LIN {X 55.470,Y -41.308,Z -105.429,A -90.000,B 90.000,C 0.000} C_DIS
LIN {X 55.184,Y -41.308,Z -107.179,A -90.000,B 90.000,C 0.000} C_DIS
LIN {X 54.822,Y -41.308,Z -109.208,A -90.000,B 90.000,C 0.000} C_DIS
LIN {X 54.818,Y -41.308,Z -109.239,A -90.000,B 90.000,C 0.000} C_DIS
LIN {X 54.778,Y -41.308,Z -109.421,A -90.000,B 90.000,C 0.000} C_DIS
LIN {X 54.161,Y -41.308,Z -111.953,A -90.000,B 90.000,C 0.000} C_DIS
LIN {X 54.080,Y -41.308,Z -112.260,A -90.000,B 90.000,C 0.000} C_DIS
LIN {X 53.759,Y -41.308,Z -113.325,A -90.000,B 90.000,C 0.000} C_DIS
LIN {X 53.214,Y -41.308,Z -114.975,A -90.000,B 90.000,C 0.000} C_DIS
LIN {X 52.425,Y -41.308,Z -117.091,A -90.000,B 90.000,C 0.000} C_DIS
LIN {X 52.337,Y -41.308,Z -117.306,A -90.000,B 90.000,C 0.000} C_DIS
LIN {X 51.749,Y -41.308,Z -118.611,A -90.000,B 90.000,C 0.000} C_DIS
LIN {X 50.611,Y -41.308,Z -120.952,A -90.000,B 90.000,C 0.000} C_DIS
LIN {X 50.435,Y -41.308,Z -121.257,A -90.000,B 90.000,C 0.000} C_DIS
LIN {X 50.184,Y -41.308,Z -121.664,A -90.000,B 90.000,C 0.000} C_DIS
LIN {X 48.891,Y -41.308,Z -123.634,A -90.000,B 90.000,C 0.000} C_DIS
LIN {X 48.351,Y -41.308,Z -124.452,A -90.000,B 90.000,C 0.000} C_DIS
LIN {X 48.205,Y -41.308,Z -124.659,A -90.000,B 90.000,C 0.000} C_DIS
LIN {X 47.984,Y -41.308,Z -124.939,A -90.000,B 90.000,C 0.000} C_DIS
LIN {X 45.252,Y -41.308,Z -127.931,A -90.000,B 90.000,C 0.000} C_DIS
LIN {X 44.992,Y -41.308,Z -128.179,A -90.000,B 90.000,C 0.000} C_DIS
LIN {X 44.294,Y -41.308,Z -128.821,A -90.000,B 90.000,C 0.000} C_DIS
LIN {X 41.919,Y -41.308,Z -130.899,A -90.000,B 90.000,C 0.000} C_DIS
LIN {X 40.833,Y -41.308,Z -131.772,A -90.000,B 90.000,C 0.000} C_DIS
LIN {X 38.770,Y -41.308,Z -133.337,A -90.000,B 90.000,C 0.000} C_DIS
LIN {X 37.043,Y -41.308,Z -134.633,A -90.000,B 90.000,C 0.000} C_DIS
LIN {X 35.762,Y -41.308,Z -135.589,A -90.000,B 90.000,C 0.000} C_DIS
LIN {X 35.411,Y -41.308,Z -135.838,A -90.000,B 90.000,C 0.000} C_DIS
LIN {X 33.546,Y -41.308,Z -137.240,A -90.000,B 90.000,C 0.000} C_DIS
LIN {X 32.468,Y -41.308,Z -138.041,A -90.000,B 90.000,C 0.000} C_DIS
LIN {X 32.425,Y -41.308,Z -138.076,A -90.000,B 90.000,C 0.000} C_DIS
LIN {X 29.828,Y -41.308,Z -139.893,A -90.000,B 90.000,C 0.000} C_DIS
LIN {X 29.382,Y -41.308,Z -140.233,A -90.000,B 90.000,C 0.000} C_DIS
LIN {X 26.864,Y -41.308,Z -141.816,A -90.000,B 90.000,C 0.000} C_DIS
LIN {X 26.120,Y -41.308,Z -142.310,A -90.000,B 90.000,C 0.000} C_DIS
LIN {X 25.779,Y -41.308,Z -142.524,A -90.000,B 90.000,C 0.000} C_DIS
LIN {X 22.899,Y -41.308,Z -144.036,A -90.000,B 90.000,C 0.000} C_DIS
LIN {X 21.842,Y -41.308,Z -144.586,A -90.000,B 90.000,C 0.000} C_DIS
LIN {X 21.477,Y -41.308,Z -144.756,A -90.000,B 90.000,C 0.000} C_DIS
LIN {X 18.835,Y -41.308,Z -145.707,A -90.000,B 90.000,C 0.000} C_DIS
LIN {X 16.834,Y -41.308,Z -146.406,A -90.000,B 90.000,C 0.000} C_DIS
LIN {X 15.872,Y -41.308,Z -146.709,A -90.000,B 90.000,C 0.000} C_DIS
LIN {X 11.057,Y -41.308,Z -147.911,A -90.000,B 90.000,C 0.000} C_DIS
LIN {X 10.662,Y -41.308,Z -147.987,A -90.000,B 90.000,C 0.000} C_DIS
LIN {X 9.668,Y -41.308,Z -148.138,A -90.000,B 90.000,C 0.000} C_DIS
LIN {X 7.179,Y -41.308,Z -148.500,A -90.000,B 90.000,C 0.000} C_DIS
LIN {X 6.274,Y -41.308,Z -148.619,A -90.000,B 90.000,C 0.000} C_DIS
LIN {X 5.872,Y -41.308,Z -148.645,A -90.000,B 90.000,C 0.000} C_DIS
LIN {X 3.525,Y -41.308,Z -148.708,A -90.000,B 90.000,C 0.000} C_DIS
LIN {X 1.800,Y -41.308,Z -148.737,A -90.000,B 90.000,C 0.000} C_DIS
LIN {X 1.354,Y -41.308,Z -148.715,A -90.000,B 90.000,C 0.000} C_DIS
LIN {X 0.760,Y -41.308,Z -148.643,A -90.000,B 90.000,C 0.000} C_DIS
LIN {X -2.452,Y -41.308,Z -148.225,A -90.000,B 90.000,C 0.000} C_DIS
LIN {X -2.823,Y -41.308,Z -148.163,A -90.000,B 90.000,C 0.000} C_DIS
LIN {X -3.340,Y -41.308,Z -148.020,A -90.000,B 90.000,C 0.000} C_DIS
LIN {X -6.560,Y -41.308,Z -147.123,A -90.000,B 90.000,C 0.000} C_DIS
LIN {X -6.893,Y -41.308,Z -147.020,A -90.000,B 90.000,C 0.000} C_DIS
LIN {X -6.944,Y -41.308,Z -147.001,A -90.000,B 90.000,C 0.000} C_DIS
LIN {X -10.523,Y -41.308,Z -145.460,A -90.000,B 90.000,C 0.000} C_DIS
LIN {X -10.889,Y -41.308,Z -145.291,A -90.000,B 90.000,C 0.000} C_DIS
LIN {X -14.025,Y -41.308,Z -143.432,A -90.000,B 90.000,C 0.000} C_DIS
LIN {X -14.270,Y -41.308,Z -143.286,A -90.000,B 90.000,C 0.000} C_DIS
LIN {X -14.609,Y -41.308,Z -143.075,A -90.000,B 90.000,C 0.000} C_DIS
LIN {X -16.177,Y -41.308,Z -141.857,A -90.000,B 90.000,C 0.000} C_DIS
LIN {X -16.469,Y -41.308,Z -141.615,A -90.000,B 90.000,C 0.000} C_DIS
LIN {X -17.822,Y -41.308,Z -140.483,A -90.000,B 90.000,C 0.000} C_DIS
LIN {X -18.130,Y -41.308,Z -140.162,A -90.000,B 90.000,C 0.000} C_DIS
LIN {X -19.708,Y -41.308,Z -138.424,A -90.000,B 90.000,C 0.000} C_DIS
LIN {X -20.576,Y -41.308,Z -137.390,A -90.000,B 90.000,C 0.000} C_DIS
LIN {X -21.291,Y -41.308,Z -136.400,A -90.000,B 90.000,C 0.000} C_DIS
LIN {X -21.957,Y -41.308,Z -135.414,A -90.000,B 90.000,C 0.000} C_DIS
LIN {X -22.580,Y -41.308,Z -134.443,A -90.000,B 90.000,C 0.000} C_DIS
LIN {X -22.732,Y -41.308,Z -134.187,A -90.000,B 90.000,C 0.000} C_DIS
LIN {X -22.837,Y -41.308,Z -133.977,A -90.000,B 90.000,C 0.000} C_DIS
LIN {X -23.185,Y -41.308,Z -133.168,A -90.000,B 90.000,C 0.000} C_DIS
LIN {X -23.761,Y -41.308,Z -131.694,A -90.000,B 90.000,C 0.000} C_DIS
LIN {X -24.464,Y -41.308,Z -129.749,A -90.000,B 90.000,C 0.000} C_DIS
LIN {X -25.043,Y -41.308,Z -128.392,A -90.000,B 90.000,C 0.000} C_DIS
LIN {X -25.131,Y -41.308,Z -128.124,A -90.000,B 90.000,C 0.000} C_DIS
LIN {X -25.348,Y -41.308,Z -127.339,A -90.000,B 90.000,C 0.000} C_DIS
LIN {X -25.372,Y -41.308,Z -127.242,A -90.000,B 90.000,C 0.000} C_DIS
LIN {X -25.461,Y -41.308,Z -126.952,A -90.000,B 90.000,C 0.000} C_DIS
LIN {X -25.852,Y -41.308,Z -125.600,A -90.000,B 90.000,C 0.000} C_DIS
LIN {X -26.676,Y -41.308,Z -123.642,A -90.000,B 90.000,C 0.000} C_DIS
LIN {X -26.686,Y -41.308,Z -123.614,A -90.000,B 90.000,C 0.000} C_DIS
LIN {X -27.017,Y -41.308,Z -122.593,A -90.000,B 90.000,C 0.000} C_DIS
LIN {X -27.366,Y -41.308,Z -121.308,A -90.000,B 90.000,C 0.000} C_DIS
LIN {X -28.113,Y -41.308,Z -119.627,A -90.000,B 90.000,C 0.000} C_DIS
LIN {X -28.235,Y -41.308,Z -119.250,A -90.000,B 90.000,C 0.000} C_DIS
LIN {X -28.388,Y -41.308,Z -118.667,A -90.000,B 90.000,C 0.000} C_DIS
LIN {X -28.690,Y -41.308,Z -117.442,A -90.000,B 90.000,C 0.000} C_DIS
LIN {X -29.303,Y -41.308,Z -115.983,A -90.000,B 90.000,C 0.000} C_DIS
LIN {X -29.504,Y -41.308,Z -115.461,A -90.000,B 90.000,C 0.000} C_DIS
LIN {X -29.584,Y -41.308,Z -115.228,A -90.000,B 90.000,C 0.000} C_DIS
LIN {X -29.707,Y -41.308,Z -114.737,A -90.000,B 90.000,C 0.000} C_DIS
LIN {X -29.745,Y -41.308,Z -114.458,A -90.000,B 90.000,C 0.000} C_DIS
LIN {X -29.886,Y -41.308,Z -113.388,A -90.000,B 90.000,C 0.000} C_DIS
LIN {X -30.064,Y -41.308,Z -112.621,A -90.000,B 90.000,C 0.000} C_DIS
LIN {X -30.103,Y -41.308,Z -112.334,A -90.000,B 90.000,C 0.000} C_DIS
LIN {X -30.199,Y -41.308,Z -111.305,A -90.000,B 90.000,C 0.000} C_DIS
LIN {X -30.447,Y -41.308,Z -109.725,A -90.000,B 90.000,C 0.000} C_DIS
LIN {X -30.483,Y -41.308,Z -109.465,A -90.000,B 90.000,C 0.000} C_DIS
LIN {X -30.496,Y -41.308,Z -109.337,A -90.000,B 90.000,C 0.000} C_DIS
LIN {X -30.516,Y -41.308,Z -109.074,A -90.000,B 90.000,C 0.000} C_DIS
LIN {X -30.504,Y -41.308,Z -108.792,A -90.000,B 90.000,C 0.000} C_DIS
LIN {X -30.411,Y -41.308,Z -107.326,A -90.000,B 90.000,C 0.000} C_DIS
LIN {X -30.397,Y -41.308,Z -106.865,A -90.000,B 90.000,C 0.000} C_DIS
LIN {X -30.386,Y -41.308,Z -106.583,A -90.000,B 90.000,C 0.000} C_DIS
LIN {X -30.285,Y -41.308,Z -105.447,A -90.000,B 90.000,C 0.000} C_DIS
LIN {X -30.192,Y -41.308,Z -104.049,A -90.000,B 90.000,C 0.000} C_DIS
LIN {X -30.163,Y -41.308,Z -103.694,A -90.000,B 90.000,C 0.000} C_DIS
LIN {X -30.120,Y -41.308,Z -102.956,A -90.000,B 90.000,C 0.000} C_DIS
LIN {X -29.985,Y -41.308,Z -101.652,A -90.000,B 90.000,C 0.000} C_DIS
LIN {X -29.637,Y -41.308,Z -99.930,A -90.000,B 90.000,C 0.000} C_DIS
LIN {X -29.511,Y -41.308,Z -99.218,A -90.000,B 90.000,C 0.000} C_DIS
LIN {X -29.260,Y -41.308,Z -98.222,A -90.000,B 90.000,C 0.000} C_DIS
LIN {X -28.951,Y -41.308,Z -96.846,A -90.000,B 90.000,C 0.000} C_DIS
LIN {X -28.873,Y -41.308,Z -96.536,A -90.000,B 90.000,C 0.000} C_DIS
LIN {X -28.764,Y -41.308,Z -96.217,A -90.000,B 90.000,C 0.000} C_DIS
LIN {X -28.435,Y -41.308,Z -95.161,A -90.000,B 90.000,C 0.000} C_DIS
LIN {X -28.154,Y -41.308,Z -94.354,A -90.000,B 90.000,C 0.000} C_DIS
LIN {X -28.113,Y -41.308,Z -94.248,A -90.000,B 90.000,C 0.000} C_DIS
LIN {X -28.028,Y -41.308,Z -94.049,A -90.000,B 90.000,C 0.000} C_DIS
LIN {X -27.020,Y -41.308,Z -91.931,A -90.000,B 90.000,C 0.000} C_DIS
LIN {X -26.081,Y -41.308,Z -90.359,A -90.000,B 90.000,C 0.000} C_DIS
LIN {X -25.839,Y -41.308,Z -89.921,A -90.000,B 90.000,C 0.000} C_DIS
LIN {X -25.669,Y -41.308,Z -89.651,A -90.000,B 90.000,C 0.000} C_DIS
LIN {X -24.410,Y -41.308,Z -87.880,A -90.000,B 90.000,C 0.000} C_DIS
LIN {X -24.228,Y -41.308,Z -87.636,A -90.000,B 90.000,C 0.000} C_DIS
LIN {X -23.011,Y -41.308,Z -86.221,A -90.000,B 90.000,C 0.000} C_DIS
LIN {X -22.429,Y -41.308,Z -85.576,A -90.000,B 90.000,C 0.000} C_DIS
LIN {X -22.261,Y -41.308,Z -85.395,A -90.000,B 90.000,C 0.000} C_DIS
LIN {X -21.069,Y -41.308,Z -84.189,A -90.000,B 90.000,C 0.000} C_DIS
LIN {X -20.042,Y -41.308,Z -83.242,A -90.000,B 90.000,C 0.000} C_DIS
LIN {X -19.639,Y -41.308,Z -82.906,A -90.000,B 90.000,C 0.000} C_DIS
LIN {X -19.414,Y -41.308,Z -82.736,A -90.000,B 90.000,C 0.000} C_DIS
LIN {X -18.873,Y -41.308,Z -82.338,A -90.000,B 90.000,C 0.000} C_DIS
LIN {X -17.806,Y -41.308,Z -81.628,A -90.000,B 90.000,C 0.000} C_DIS
LIN {X -16.939,Y -41.308,Z -81.143,A -90.000,B 90.000,C 0.000} C_DIS
LIN {X -16.688,Y -41.308,Z -81.016,A -90.000,B 90.000,C 0.000} C_DIS
LIN {X -15.805,Y -41.308,Z -80.619,A -90.000,B 90.000,C 0.000} C_DIS
LIN {X -14.901,Y -41.308,Z -80.303,A -90.000,B 90.000,C 0.000} C_DIS
LIN {X -13.548,Y -41.308,Z -79.901,A -90.000,B 90.000,C 0.000} C_DIS
LIN {X -12.288,Y -41.308,Z -79.649,A -90.000,B 90.000,C 0.000} C_DIS
LIN {X -12.008,Y -41.308,Z -79.617,A -90.000,B 90.000,C 0.000} C_DIS
LIN {X -11.056,Y -41.308,Z -79.521,A -90.000,B 90.000,C 0.000} C_DIS
LIN {X -10.367,Y -41.308,Z -79.494,A -90.000,B 90.000,C 0.000} C_DIS
LIN {X -8.489,Y -41.308,Z -79.501,A -90.000,B 90.000,C 0.000} C_DIS
LIN {X -5.734,Y -41.308,Z -79.670,A -90.000,B 90.000,C 0.000} C_DIS
LIN {X -5.452,Y -41.308,Z -79.690,A -90.000,B 90.000,C 0.000} C_DIS
LIN {X -4.926,Y -41.308,Z -79.755,A -90.000,B 90.000,C 0.000} C_DIS
LIN {X -3.458,Y -41.308,Z -79.966,A -90.000,B 90.000,C 0.000} C_DIS
LIN {X -2.097,Y -41.308,Z -80.208,A -90.000,B 90.000,C 0.000} C_DIS
LIN {X -1.466,Y -41.308,Z -80.327,A -90.000,B 90.000,C 0.000} C_DIS
LIN {X 0.990,Y -41.308,Z -80.823,A -90.000,B 90.000,C 0.000} C_DIS
LIN {X 2.920,Y -41.308,Z -81.243,A -90.000,B 90.000,C 0.000} C_DIS
LIN {X 3.999,Y -41.308,Z -81.474,A -90.000,B 90.000,C 0.000} C_DIS
LIN {X 6.583,Y -41.308,Z -82.083,A -90.000,B 90.000,C 0.000} C_DIS
LIN {X 7.278,Y -41.308,Z -82.255,A -90.000,B 90.000,C 0.000} C_DIS
LIN {X 9.781,Y -41.308,Z -82.880,A -90.000,B 90.000,C 0.000} C_DIS
LIN {X 10.695,Y -41.308,Z -83.134,A -90.000,B 90.000,C 0.000} C_DIS
LIN {X 12.282,Y -41.308,Z -83.509,A -90.000,B 90.000,C 0.000} C_DIS
LIN {X 12.596,Y -41.308,Z -83.584,A -90.000,B 90.000,C 0.000} C_DIS
LIN {X 13.574,Y -41.308,Z -83.847,A -90.000,B 90.000,C 0.000} C_DIS
LIN {X 14.545,Y -41.308,Z -84.040,A -90.000,B 90.000,C 0.000} C_DIS
LIN {X 16.321,Y -41.308,Z -84.427,A -90.000,B 90.000,C 0.000} C_DIS
LIN {X 16.721,Y -41.308,Z -84.484,A -90.000,B 90.000,C 0.000} C_DIS
LIN {X 17.318,Y -41.308,Z -84.561,A -90.000,B 90.000,C 0.000} C_DIS
LIN {X 18.860,Y -41.308,Z -84.755,A -90.000,B 90.000,C 0.000} C_DIS
LIN {X 19.195,Y -41.308,Z -84.791,A -90.000,B 90.000,C 0.000} C_DIS
LIN {X 20.625,Y -41.308,Z -84.831,A -90.000,B 90.000,C 0.000} C_DIS
LIN {X 21.068,Y -41.308,Z -84.812,A -90.000,B 90.000,C 0.000} C_DIS
LIN {X 21.675,Y -41.308,Z -84.762,A -90.000,B 90.000,C 0.000} C_DIS
LIN {X 22.544,Y -41.308,Z -84.619,A -90.000,B 90.000,C 0.000} C_DIS
LIN {X 22.792,Y -41.308,Z -84.576,A -90.000,B 90.000,C 0.000} C_DIS
LIN {X 23.921,Y -41.308,Z -84.001,A -90.000,B 90.000,C 0.000} C_DIS
LIN {X 24.234,Y -41.308,Z -83.731,A -90.000,B 90.000,C 0.000} C_DIS
LIN {X 25.145,Y -41.308,Z -82.984,A -90.000,B 90.000,C 0.000} C_DIS
LIN {X 26.310,Y -41.308,Z -81.865,A -90.000,B 90.000,C 0.000} C_DIS
LIN {X 26.500,Y -41.308,Z -81.723,A -90.000,B 90.000,C 0.000} C_DIS
LIN {X 27.217,Y -41.308,Z -81.212,A -90.000,B 90.000,C 0.000} C_DIS
LIN {X 27.880,Y -41.308,Z -80.766,A -90.000,B 90.000,C 0.000} C_DIS
LIN {X 28.606,Y -41.308,Z -80.372,A -90.000,B 90.000,C 0.000} C_DIS
LIN {X 28.858,Y -41.308,Z -80.245,A -90.000,B 90.000,C 0.000} C_DIS
LIN {X 32.394,Y -41.308,Z -78.944,A -90.000,B 90.000,C 0.000} C_DIS
LIN {X 34.865,Y -41.308,Z -78.150,A -90.000,B 90.000,C 0.000} C_DIS
LIN {X 36.376,Y -41.308,Z -77.574,A -90.000,B 90.000,C 0.000} C_DIS
LIN {X 36.658,Y -41.308,Z -77.445,A -90.000,B 90.000,C 0.000} C_DIS
LIN {X 36.711,Y -41.308,Z -77.406,A -90.000,B 90.000,C 0.000} C_DIS
LIN {X 36.279,Y -41.308,Z -77.381,A -90.000,B 90.000,C 0.000} C_DIS
LIN {X 35.892,Y -41.308,Z -77.401,A -90.000,B 90.000,C 0.000} C_DIS
LIN {X 35.542,Y -41.308,Z -77.370,A -90.000,B 90.000,C 0.000} C_DIS
LIN {X 34.944,Y -41.308,Z -77.302,A -90.000,B 90.000,C 0.000} C_DIS
LIN {X 34.710,Y -41.308,Z -77.248,A -90.000,B 90.000,C 0.000} C_DIS
LIN {X 34.690,Y -41.308,Z -77.245,A -90.000,B 90.000,C 0.000} C_DIS
LIN {X 34.551,Y -41.308,Z -77.209,A -90.000,B 90.000,C 0.000} C_DIS
LIN {X 34.342,Y -41.308,Z -77.160,A -90.000,B 90.000,C 0.000} C_DIS
LIN {X 34.182,Y -41.308,Z -77.145,A -90.000,B 90.000,C 0.000} C_DIS
LIN {X 33.840,Y -41.308,Z -77.064,A -90.000,B 90.000,C 0.000} C_DIS
LIN {X 33.513,Y -41.308,Z -76.935,A -90.000,B 90.000,C 0.000} C_DIS
LIN {X 33.246,Y -41.308,Z -76.821,A -90.000,B 90.000,C 0.000} C_DIS
LIN {X 33.194,Y -41.308,Z -76.802,A -90.000,B 90.000,C 0.000} C_DIS
LIN {X 32.906,Y -41.308,Z -76.688,A -90.000,B 90.000,C 0.000} C_DIS
LIN {X 32.600,Y -41.308,Z -76.515,A -90.000,B 90.000,C 0.000} C_DIS
LIN {X 32.189,Y -41.308,Z -76.218,A -90.000,B 90.000,C 0.000} C_DIS
LIN {X 32.137,Y -41.308,Z -76.188,A -90.000,B 90.000,C 0.000} C_DIS
LIN {X 32.111,Y -41.308,Z -76.168,A -90.000,B 90.000,C 0.000} C_DIS
LIN {X 31.860,Y -41.308,Z -75.973,A -90.000,B 90.000,C 0.000} C_DIS
LIN {X 31.615,Y -41.308,Z -75.720,A -90.000,B 90.000,C 0.000} C_DIS
LIN {X 31.393,Y -41.308,Z -75.413,A -90.000,B 90.000,C 0.000} C_DIS
LIN {X 31.123,Y -41.308,Z -75.016,A -90.000,B 90.000,C 0.000} C_DIS
LIN {X 30.978,Y -41.308,Z -74.811,A -90.000,B 90.000,C 0.000} C_DIS
LIN {X 30.801,Y -41.308,Z -74.476,A -90.000,B 90.000,C 0.000} C_DIS
LIN {X 30.670,Y -41.308,Z -74.120,A -90.000,B 90.000,C 0.000} C_DIS
LIN {X 30.513,Y -41.308,Z -73.557,A -90.000,B 90.000,C 0.000} C_DIS
LIN {X 30.454,Y -41.308,Z -73.158,A -90.000,B 90.000,C 0.000} C_DIS
LIN {X 30.401,Y -41.308,Z -72.580,A -90.000,B 90.000,C 0.000} C_DIS
LIN {X 30.402,Y -41.308,Z -72.545,A -90.000,B 90.000,C 0.000} C_DIS
LIN {X 30.356,Y -41.308,Z -71.582,A -90.000,B 90.000,C 0.000} C_DIS
LIN {X 30.352,Y -41.308,Z -71.406,A -90.000,B 90.000,C 0.000} C_DIS
LIN {X 30.362,Y -41.308,Z -70.965,A -90.000,B 90.000,C 0.000} C_DIS
LIN {X 30.411,Y -41.308,Z -70.384,A -90.000,B 90.000,C 0.000} C_DIS
LIN {X 30.466,Y -41.308,Z -69.932,A -90.000,B 90.000,C 0.000} C_DIS
LIN {X 30.522,Y -41.308,Z -69.610,A -90.000,B 90.000,C 0.000} C_DIS
LIN {X 30.577,Y -41.308,Z -69.206,A -90.000,B 90.000,C 0.000} C_DIS
LIN {X 30.488,Y -41.308,Z -68.758,A -90.000,B 90.000,C 0.000} C_DIS
LIN {X 30.479,Y -41.308,Z -68.643,A -90.000,B 90.000,C 0.000} C_DIS
LIN {X 30.465,Y -41.308,Z -68.403,A -90.000,B 90.000,C 0.000} C_DIS
LIN {X 30.441,Y -41.308,Z -68.159,A -90.000,B 90.000,C 0.000} C_DIS
LIN {X 30.373,Y -41.308,Z -67.312,A -90.000,B 90.000,C 0.000} C_DIS
LIN {X 30.356,Y -41.308,Z -67.021,A -90.000,B 90.000,C 0.000} C_DIS
LIN {X 30.378,Y -41.308,Z -66.364,A -90.000,B 90.000,C 0.000} C_DIS
LIN {X 30.428,Y -41.308,Z -65.571,A -90.000,B 90.000,C 0.000} C_DIS
LIN {X 30.458,Y -41.308,Z -65.229,A -90.000,B 90.000,C 0.000} C_DIS
LIN {X 30.652,Y -41.308,Z -64.365,A -90.000,B 90.000,C 0.000} C_DIS
LIN {X 30.731,Y -41.308,Z -64.056,A -90.000,B 90.000,C 0.000} C_DIS
LIN {X 30.846,Y -41.308,Z -63.730,A -90.000,B 90.000,C 0.000} C_DIS
LIN {X 30.869,Y -41.308,Z -63.646,A -90.000,B 90.000,C 0.000} C_DIS
LIN {X 30.956,Y -41.308,Z -63.430,A -90.000,B 90.000,C 0.000} C_DIS
LIN {X 31.055,Y -41.308,Z -63.200,A -90.000,B 90.000,C 0.000} C_DIS
LIN {X 31.221,Y -41.308,Z -62.936,A -90.000,B 90.000,C 0.000} C_DIS
LIN {X 31.433,Y -41.308,Z -62.669,A -90.000,B 90.000,C 0.000} C_DIS
LIN {X 31.625,Y -41.308,Z -62.462,A -90.000,B 90.000,C 0.000} C_DIS
LIN {X 31.850,Y -41.308,Z -62.293,A -90.000,B 90.000,C 0.000} C_DIS
LIN {X 31.898,Y -41.308,Z -62.269,A -90.000,B 90.000,C 0.000} C_DIS
LIN {X 31.934,Y -41.308,Z -62.101,A -90.000,B 90.000,C 0.000} C_DIS
LIN {X 32.239,Y -41.308,Z -60.873,A -90.000,B 90.000,C 0.000} C_DIS
LIN {X 32.373,Y -41.308,Z -60.427,A -90.000,B 90.000,C 0.000} C_DIS
LIN {X 32.524,Y -41.308,Z -59.945,A -90.000,B 90.000,C 0.000} C_DIS
LIN {X 32.690,Y -41.308,Z -59.445,A -90.000,B 90.000,C 0.000} C_DIS
LIN {X 32.902,Y -41.308,Z -58.788,A -90.000,B 90.000,C 0.000} C_DIS
LIN {X 33.082,Y -41.308,Z -58.320,A -90.000,B 90.000,C 0.000} C_DIS
LIN {X 33.134,Y -41.308,Z -58.190,A -90.000,B 90.000,C 0.000} C_DIS
LIN {X 33.292,Y -41.308,Z -57.823,A -90.000,B 90.000,C 0.000} C_DIS
LIN {X 33.489,Y -41.308,Z -57.449,A -90.000,B 90.000,C 0.000} C_DIS
LIN {X 33.657,Y -41.308,Z -57.144,A -90.000,B 90.000,C 0.000} C_DIS
LIN {X 33.822,Y -41.308,Z -56.825,A -90.000,B 90.000,C 0.000} C_DIS
LIN {X 33.949,Y -41.308,Z -56.585,A -90.000,B 90.000,C 0.000} C_DIS
LIN {X 34.158,Y -41.308,Z -56.223,A -90.000,B 90.000,C 0.000} C_DIS
LIN {X 34.385,Y -41.308,Z -55.890,A -90.000,B 90.000,C 0.000} C_DIS
LIN {X 34.487,Y -41.308,Z -55.759,A -90.000,B 90.000,C 0.000} C_DIS
LIN {X 34.847,Y -41.308,Z -55.337,A -90.000,B 90.000,C 0.000} C_DIS
LIN {X 34.935,Y -41.308,Z -55.224,A -90.000,B 90.000,C 0.000} C_DIS
LIN {X 35.201,Y -41.308,Z -54.922,A -90.000,B 90.000,C 0.000} C_DIS
LIN {X 35.609,Y -41.308,Z -54.560,A -90.000,B 90.000,C 0.000} C_DIS
LIN {X 35.931,Y -41.308,Z -54.296,A -90.000,B 90.000,C 0.000} C_DIS
LIN {X 36.272,Y -41.308,Z -54.006,A -90.000,B 90.000,C 0.000} C_DIS
LIN {X 36.584,Y -41.308,Z -53.791,A -90.000,B 90.000,C 0.000} C_DIS
LIN {X 36.921,Y -41.308,Z -53.618,A -90.000,B 90.000,C 0.000} C_DIS
LIN {X 37.709,Y -41.308,Z -53.229,A -90.000,B 90.000,C 0.000} C_DIS
LIN {X 38.066,Y -41.308,Z -53.102,A -90.000,B 90.000,C 0.000} C_DIS
LIN {X 38.437,Y -41.308,Z -53.023,A -90.000,B 90.000,C 0.000} C_DIS
LIN {X 38.700,Y -41.308,Z -52.974,A -90.000,B 90.000,C 0.000} C_DIS
LIN {X 39.354,Y -41.308,Z -52.862,A -90.000,B 90.000,C 0.000} C_DIS
LIN {X 39.731,Y -41.308,Z -52.832,A -90.000,B 90.000,C 0.000} C_DIS
LIN {X 40.110,Y -41.308,Z -52.853,A -90.000,B 90.000,C 0.000} C_DIS
LIN {X 41.155,Y -41.308,Z -52.980,A -90.000,B 90.000,C 0.000} C_DIS
LIN {X 41.602,Y -41.308,Z -53.047,A -90.000,B 90.000,C 0.000} C_DIS
LIN {X 41.990,Y -41.308,Z -53.154,A -90.000,B 90.000,C 0.000} C_DIS
LIN {X 42.647,Y -41.308,Z -53.423,A -90.000,B 90.000,C 0.000} C_DIS
LIN {X 42.780,Y -41.308,Z -53.478,A -90.000,B 90.000,C 0.000} C_DIS
LIN {X 43.521,Y -41.308,Z -53.797,A -90.000,B 90.000,C 0.000} C_DIS
LIN {X 44.003,Y -41.308,Z -54.036,A -90.000,B 90.000,C 0.000} C_DIS
LIN {X 44.849,Y -41.308,Z -54.524,A -90.000,B 90.000,C 0.000} C_DIS
LIN {X 45.045,Y -41.308,Z -54.659,A -90.000,B 90.000,C 0.000} C_DIS
LIN {X 45.065,Y -41.308,Z -54.675,A -90.000,B 90.000,C 0.000} C_DIS
LIN {X 45.358,Y -41.308,Z -54.860,A -90.000,B 90.000,C 0.000} C_DIS
LIN {X 45.811,Y -41.308,Z -55.153,A -90.000,B 90.000,C 0.000} C_DIS
LIN {X 46.165,Y -41.308,Z -55.299,A -90.000,B 90.000,C 0.000} C_DIS
LIN {X 46.737,Y -41.308,Z -55.294,A -90.000,B 90.000,C 0.000} C_DIS
LIN {X 47.010,Y -41.308,Z -55.260,A -90.000,B 90.000,C 0.000} C_DIS
LIN {X 47.961,Y -41.308,Z -55.134,A -90.000,B 90.000,C 0.000} C_DIS
LIN {X 48.312,Y -41.308,Z -55.112,A -90.000,B 90.000,C 0.000} C_DIS
LIN {X 48.661,Y -41.308,Z -55.117,A -90.000,B 90.000,C 0.000} C_DIS
LIN {X 49.862,Y -41.308,Z -55.125,A -90.000,B 90.000,C 0.000} C_DIS
LIN {X 50.212,Y -41.308,Z -55.152,A -90.000,B 90.000,C 0.000} C_DIS
LIN {X 50.555,Y -41.308,Z -55.228,A -90.000,B 90.000,C 0.000} C_DIS
LIN {X 50.995,Y -41.308,Z -55.386,A -90.000,B 90.000,C 0.000} C_DIS
LIN {X 52.266,Y -41.308,Z -55.813,A -90.000,B 90.000,C 0.000} C_DIS
LIN {X 52.594,Y -41.308,Z -55.937,A -90.000,B 90.000,C 0.000} C_DIS
LIN {X 52.902,Y -41.308,Z -56.107,A -90.000,B 90.000,C 0.000} C_DIS
LIN {X 53.274,Y -41.308,Z -56.363,A -90.000,B 90.000,C 0.000} C_DIS
LIN {X 54.616,Y -41.308,Z -57.527,A -90.000,B 90.000,C 0.000} C_DIS
LIN {X 55.075,Y -41.308,Z -57.901,A -90.000,B 90.000,C 0.000} C_DIS
LIN {X 55.361,Y -41.308,Z -58.149,A -90.000,B 90.000,C 0.000} C_DIS
LIN {X 55.613,Y -41.308,Z -58.433,A -90.000,B 90.000,C 0.000} C_DIS
LIN {X 56.273,Y -41.308,Z -59.243,A -90.000,B 90.000,C 0.000} C_DIS
LIN {X 56.836,Y -41.308,Z -60.063,A -90.000,B 90.000,C 0.000} C_DIS
LIN {X 57.249,Y -41.308,Z -60.739,A -90.000,B 90.000,C 0.000} C_DIS
LIN {X 57.417,Y -41.308,Z -61.048,A -90.000,B 90.000,C 0.000} C_DIS
LIN {X 57.694,Y -41.308,Z -61.603,A -90.000,B 90.000,C 0.000} C_DIS
LIN {X 58.519,Y -41.308,Z -63.268,A -90.000,B 90.000,C 0.000} C_DIS
LIN {X 58.625,Y -41.308,Z -63.485,A -90.000,B 90.000,C 0.000} C_DIS
LIN {X 58.747,Y -41.308,Z -63.814,A -90.000,B 90.000,C 0.000} C_DIS
LIN {X 58.855,Y -41.308,Z -64.192,A -90.000,B 90.000,C 0.000} C_DIS
LIN {X 59.303,Y -41.308,Z -65.629,A -90.000,B 90.000,C 0.000} C_DIS
LIN {X 59.469,Y -41.308,Z -66.070,A -90.000,B 90.000,C 0.000} C_DIS
LIN {X 59.522,Y -41.308,Z -66.215,A -90.000,B 90.000,C 0.000} C_DIS
LIN {X 59.609,Y -41.308,Z -66.491,A -90.000,B 90.000,C 0.000} C_DIS
LIN {X 59.684,Y -41.308,Z -66.801,A -90.000,B 90.000,C 0.000} C_DIS
LIN {X 59.736,Y -41.308,Z -67.319,A -90.000,B 90.000,C 0.000} C_DIS
LIN {X 59.960,Y -41.308,Z -68.158,A -90.000,B 90.000,C 0.000} C_DIS
LIN {X 59.981,Y -41.308,Z -68.224,A -90.000,B 90.000,C 0.000} C_DIS
LIN {X 60.005,Y -41.308,Z -68.266,A -90.000,B 90.000,C 0.000} C_DIS
LIN {X 60.306,Y -41.308,Z -68.917,A -90.000,B 90.000,C 0.000} C_DIS
LIN {X 60.380,Y -41.308,Z -69.189,A -90.000,B 90.000,C 0.000} C_DIS
LIN {X 60.405,Y -41.308,Z -69.470,A -90.000,B 90.000,C 0.000} C_DIS
LIN {X 60.440,Y -41.308,Z -69.915,A -90.000,B 90.000,C 0.000} C_DIS
LIN {X 60.841,Y -41.308,Z -70.835,A -90.000,B 90.000,C 0.000} C_DIS
LIN {X 61.105,Y -41.308,Z -71.199,A -90.000,B 90.000,C 0.000} C_DIS
LIN {X 61.224,Y -41.308,Z -71.405,A -90.000,B 90.000,C 0.000} C_DIS
LIN {X 61.297,Y -41.308,Z -71.629,A -90.000,B 90.000,C 0.000} C_DIS
LIN {X 61.343,Y -41.308,Z -71.804,A -90.000,B 90.000,C 0.000} C_DIS
LIN {X 61.380,Y -41.308,Z -71.952,A -90.000,B 90.000,C 0.000} C_DIS
LIN {X 61.405,Y -41.308,Z -72.132,A -90.000,B 90.000,C 0.000} C_DIS
LIN {X 61.391,Y -41.308,Z -72.602,A -90.000,B 90.000,C 0.000} C_DIS
LIN {X 61.868,Y -41.308,Z -73.402,A -90.000,B 90.000,C 0.000} C_DIS
LIN {X 61.932,Y -41.308,Z -73.517,A -90.000,B 90.000,C 0.000} C_DIS
LIN {X 63.002,Y -41.308,Z -74.385,A -90.000,B 90.000,C 0.000} C_DIS
LIN {X 63.117,Y -41.308,Z -74.523,A -90.000,B 90.000,C 0.000} C_DIS
LIN {X 63.613,Y -41.308,Z -75.176,A -90.000,B 90.000,C 0.000} C_DIS
LIN {X 65.360,Y -41.308,Z -75.761,A -90.000,B 90.000,C 0.000} C_DIS
LIN {X 66.354,Y -41.308,Z -76.243,A -90.000,B 90.000,C 0.000} C_DIS
LIN {X 66.836,Y -41.308,Z -76.513,A -90.000,B 90.000,C 0.000} C_DIS
LIN {X 67.028,Y -41.308,Z -76.651,A -90.000,B 90.000,C 0.000} C_DIS
LIN {X 67.842,Y -41.308,Z -77.413,A -90.000,B 90.000,C 0.000} C_DIS
LIN {X 68.116,Y -41.308,Z -77.674,A -90.000,B 90.000,C 0.000} C_DIS
LIN {X 69.042,Y -41.308,Z -77.886,A -90.000,B 90.000,C 0.000} C_DIS
LIN {X 69.260,Y -41.308,Z -77.981,A -90.000,B 90.000,C 0.000} C_DIS
LIN {X 69.975,Y -41.308,Z -78.474,A -90.000,B 90.000,C 0.000} C_DIS
LIN {X 70.587,Y -41.308,Z -79.076,A -90.000,B 90.000,C 0.000} C_DIS
LIN {X 70.966,Y -41.308,Z -79.296,A -90.000,B 90.000,C 0.000} C_DIS
LIN {X 71.203,Y -41.308,Z -79.458,A -90.000,B 90.000,C 0.000} C_DIS
LIN {X 71.433,Y -41.308,Z -79.654,A -90.000,B 90.000,C 0.000} C_DIS
LIN {X 71.631,Y -41.308,Z -79.751,A -90.000,B 90.000,C 0.000} C_DIS
LIN {X 71.864,Y -41.308,Z -79.909,A -90.000,B 90.000,C 0.000} C_DIS
LIN {X 72.573,Y -41.308,Z -80.530,A -90.000,B 90.000,C 0.000} C_DIS
LIN {X 72.588,Y -41.308,Z -80.545,A -90.000,B 90.000,C 0.000} C_DIS
LIN {X 72.622,Y -41.308,Z -80.570,A -90.000,B 90.000,C 0.000} C_DIS
LIN {X 72.886,Y -41.308,Z -80.783,A -90.000,B 90.000,C 0.000} C_DIS
LIN {X 73.118,Y -41.308,Z -80.991,A -90.000,B 90.000,C 0.000} C_DIS
LIN {X 73.252,Y -41.308,Z -81.064,A -90.000,B 90.000,C 0.000} C_DIS
LIN {X 73.340,Y -41.308,Z -81.124,A -90.000,B 90.000,C 0.000} C_DIS
LIN {X 73.932,Y -41.308,Z -81.530,A -90.000,B 90.000,C 0.000} C_DIS
LIN {X 74.076,Y -41.308,Z -81.655,A -90.000,B 90.000,C 0.000} C_DIS
LIN {X 74.183,Y -41.308,Z -81.721,A -90.000,B 90.000,C 0.000} C_DIS
LIN {X 74.570,Y -41.308,Z -82.017,A -90.000,B 90.000,C 0.000} C_DIS
LIN {X 74.701,Y -41.308,Z -82.078,A -90.000,B 90.000,C 0.000} C_DIS
LIN {X 75.295,Y -41.308,Z -82.362,A -90.000,B 90.000,C 0.000} C_DIS
LIN {X 75.636,Y -41.308,Z -82.476,A -90.000,B 90.000,C 0.000} C_DIS
LIN {X 76.345,Y -41.308,Z -82.584,A -90.000,B 90.000,C 0.000} C_DIS
LIN {X 76.385,Y -41.308,Z -82.577,A -90.000,B 90.000,C 0.000} C_DIS
LIN {X 77.209,Y -41.308,Z -82.502,A -90.000,B 90.000,C 0.000} C_DIS
LIN {X 77.471,Y -41.308,Z -82.444,A -90.000,B 90.000,C 0.000} C_DIS
LIN {X 78.012,Y -41.308,Z -82.289,A -90.000,B 90.000,C 0.000} C_DIS
LIN {X 78.258,Y -41.308,Z -82.226,A -90.000,B 90.000,C 0.000} C_DIS
LIN {X 78.430,Y -41.308,Z -82.190,A -90.000,B 90.000,C 0.000} C_DIS
LIN {X 79.273,Y -41.308,Z -81.919,A -90.000,B 90.000,C 0.000} C_DIS
LIN {X 79.827,Y -41.308,Z -81.693,A -90.000,B 90.000,C 0.000} C_DIS
LIN {X 79.937,Y -41.308,Z -81.641,A -90.000,B 90.000,C 0.000} C_DIS
LIN {X 80.363,Y -41.308,Z -81.265,A -90.000,B 90.000,C 0.000} C_DIS
LIN {X 80.545,Y -41.308,Z -80.932,A -90.000,B 90.000,C 0.000} C_DIS
LIN {X 80.667,Y -41.308,Z -80.018,A -90.000,B 90.000,C 0.000} C_DIS
LIN {X 80.636,Y -41.308,Z -79.445,A -90.000,B 90.000,C 0.000} C_DIS
LIN {X 80.627,Y -41.308,Z -79.042,A -90.000,B 90.000,C 0.000} C_DIS
LIN {X 80.636,Y -41.308,Z -78.656,A -90.000,B 90.000,C 0.000} C_DIS
LIN {X 80.610,Y -41.308,Z -78.359,A -90.000,B 90.000,C 0.000} C_DIS
LIN {X 80.571,Y -41.308,Z -77.854,A -90.000,B 90.000,C 0.000} C_DIS
LIN {X 80.431,Y -41.308,Z -76.989,A -90.000,B 90.000,C 0.000} C_DIS
LIN {X 80.387,Y -41.308,Z -76.575,A -90.000,B 90.000,C 0.000} C_DIS
LIN {X 80.334,Y -41.308,Z -76.180,A -90.000,B 90.000,C 0.000} C_DIS
LIN {X 80.270,Y -41.308,Z -75.662,A -90.000,B 90.000,C 0.000} C_DIS
LIN {X 80.193,Y -41.308,Z -75.286,A -90.000,B 90.000,C 0.000} C_DIS
LIN {X 80.055,Y -41.308,Z -74.540,A -90.000,B 90.000,C 0.000} C_DIS
LIN {X 80.040,Y -41.308,Z -74.390,A -90.000,B 90.000,C 0.000} C_DIS
LIN {X 79.912,Y -41.308,Z -73.324,A -90.000,B 90.000,C 0.000} C_DIS
LIN {X 79.847,Y -41.308,Z -72.930,A -90.000,B 90.000,C 0.000} C_DIS
LIN {X 79.751,Y -41.308,Z -72.302,A -90.000,B 90.000,C 0.000} C_DIS
LIN {X 79.707,Y -41.308,Z -71.849,A -90.000,B 90.000,C 0.000} C_DIS
LIN {X 79.696,Y -41.308,Z -71.694,A -90.000,B 90.000,C 0.000} C_DIS
LIN {X 79.678,Y -41.308,Z -71.286,A -90.000,B 90.000,C 0.000} C_DIS
LIN {X 79.671,Y -41.308,Z -70.819,A -90.000,B 90.000,C 0.000} C_DIS
LIN {X 79.671,Y -41.308,Z -70.171,A -90.000,B 90.000,C 0.000} C_DIS
LIN {X 79.685,Y -41.308,Z -69.516,A -90.000,B 90.000,C 0.000} C_DIS
LIN {X 79.709,Y -41.308,Z -69.073,A -90.000,B 90.000,C 0.000} C_DIS
LIN {X 79.750,Y -41.308,Z -68.632,A -90.000,B 90.000,C 0.000} C_DIS
LIN {X 79.821,Y -41.308,Z -68.161,A -90.000,B 90.000,C 0.000} C_DIS
LIN {X 79.981,Y -41.308,Z -67.347,A -90.000,B 90.000,C 0.000} C_DIS
LIN {X 80.177,Y -41.308,Z -66.619,A -90.000,B 90.000,C 0.000} C_DIS
LIN {X 80.342,Y -41.308,Z -66.113,A -90.000,B 90.000,C 0.000} C_DIS
LIN {X 80.540,Y -41.308,Z -65.669,A -90.000,B 90.000,C 0.000} C_DIS
LIN {X 81.017,Y -41.308,Z -64.624,A -90.000,B 90.000,C 0.000} C_DIS
LIN {X 81.207,Y -41.308,Z -64.250,A -90.000,B 90.000,C 0.000} C_DIS
LIN {X 81.438,Y -41.308,Z -63.804,A -90.000,B 90.000,C 0.000} C_DIS
LIN {X 81.708,Y -41.308,Z -63.344,A -90.000,B 90.000,C 0.000} C_DIS
LIN {X 82.705,Y -41.308,Z -61.742,A -90.000,B 90.000,C 0.000} C_DIS
LIN {X 84.243,Y -41.308,Z -59.630,A -90.000,B 90.000,C 0.000} C_DIS
LIN {X 85.732,Y -41.308,Z -57.856,A -90.000,B 90.000,C 0.000} C_DIS
LIN {X 86.059,Y -41.308,Z -57.494,A -90.000,B 90.000,C 0.000} C_DIS
LIN {X 87.795,Y -41.308,Z -55.685,A -90.000,B 90.000,C 0.000} C_DIS
LIN {X 89.901,Y -41.308,Z -53.759,A -90.000,B 90.000,C 0.000} C_DIS
LIN {X 90.156,Y -41.308,Z -53.529,A -90.000,B 90.000,C 0.000} C_DIS
LIN {X 92.336,Y -41.308,Z -51.661,A -90.000,B 90.000,C 0.000} C_DIS
LIN {X 94.367,Y -41.308,Z -49.945,A -90.000,B 90.000,C 0.000} C_DIS
LIN {X 96.070,Y -41.308,Z -48.453,A -90.000,B 90.000,C 0.000} C_DIS
LIN {X 97.648,Y -41.308,Z -46.921,A -90.000,B 90.000,C 0.000} C_DIS
LIN {X 99.081,Y -41.308,Z -45.409,A -90.000,B 90.000,C 0.000} C_DIS
LIN {X 100.198,Y -41.308,Z -44.163,A -90.000,B 90.000,C 0.000} C_DIS
LIN {X 101.129,Y -41.308,Z -43.113,A -90.000,B 90.000,C 0.000} C_DIS
LIN {X 101.593,Y -41.308,Z -42.598,A -90.000,B 90.000,C 0.000} C_DIS
LIN {X 102.507,Y -41.308,Z -41.597,A -90.000,B 90.000,C 0.000} C_DIS
LIN {X 103.068,Y -41.308,Z -41.024,A -90.000,B 90.000,C 0.000} C_DIS
LIN {X 103.316,Y -41.308,Z -40.771,A -90.000,B 90.000,C 0.000} C_DIS
LIN {X 103.675,Y -41.308,Z -40.443,A -90.000,B 90.000,C 0.000} C_DIS
LIN {X 103.973,Y -41.308,Z -40.177,A -90.000,B 90.000,C 0.000} C_DIS
LIN {X 104.471,Y -41.308,Z -39.738,A -90.000,B 90.000,C 0.000} C_DIS
LIN {X 104.833,Y -41.308,Z -39.455,A -90.000,B 90.000,C 0.000} C_DIS
LIN {X 105.188,Y -41.308,Z -39.182,A -90.000,B 90.000,C 0.000} C_DIS
LIN {X 105.612,Y -41.308,Z -38.867,A -90.000,B 90.000,C 0.000} C_DIS
LIN {X 105.910,Y -41.308,Z -38.665,A -90.000,B 90.000,C 0.000} C_DIS
LIN {X 106.316,Y -41.308,Z -38.399,A -90.000,B 90.000,C 0.000} C_DIS
LIN {X 106.878,Y -41.308,Z -38.075,A -90.000,B 90.000,C 0.000} C_DIS
LIN {X 107.285,Y -41.308,Z -37.845,A -90.000,B 90.000,C 0.000} C_DIS
LIN {X 107.391,Y -41.308,Z -37.790,A -90.000,B 90.000,C 0.000} C_DIS
LIN {X 108.215,Y -41.308,Z -37.430,A -90.000,B 90.000,C 0.000} C_DIS
LIN {X 108.398,Y -41.308,Z -37.363,A -90.000,B 90.000,C 0.000} C_DIS
LIN {X 108.825,Y -41.308,Z -37.222,A -90.000,B 90.000,C 0.000} C_DIS
LIN {X 109.037,Y -41.308,Z -37.155,A -90.000,B 90.000,C 0.000} C_DIS
LIN {X 109.465,Y -41.308,Z -37.051,A -90.000,B 90.000,C 0.000} C_DIS
LIN {X 109.533,Y -41.308,Z -37.038,A -90.000,B 90.000,C 0.000} C_DIS
LIN {X 110.241,Y -41.308,Z -36.945,A -90.000,B 90.000,C 0.000} C_DIS
LIN {X 110.401,Y -41.308,Z -36.933,A -90.000,B 90.000,C 0.000} C_DIS
LIN {X 110.691,Y -41.308,Z -36.927,A -90.000,B 90.000,C 0.000} C_DIS
LIN {X 111.285,Y -41.308,Z -36.949,A -90.000,B 90.000,C 0.000} C_DIS
LIN {X 111.402,Y -41.308,Z -36.960,A -90.000,B 90.000,C 0.000} C_DIS
LIN {X 111.725,Y -41.308,Z -37.010,A -90.000,B 90.000,C 0.000} C_DIS
LIN {X 111.887,Y -41.308,Z -37.043,A -90.000,B 90.000,C 0.000} C_DIS
LIN {X 112.040,Y -41.308,Z -37.078,A -90.000,B 90.000,C 0.000} C_DIS
LIN {X 112.502,Y -41.308,Z -37.205,A -90.000,B 90.000,C 0.000} C_DIS
LIN {X 112.921,Y -41.308,Z -37.374,A -90.000,B 90.000,C 0.000} C_DIS
LIN {X 113.493,Y -41.308,Z -37.682,A -90.000,B 90.000,C 0.000} C_DIS
LIN {X 113.591,Y -41.308,Z -37.744,A -90.000,B 90.000,C 0.000} C_DIS
LIN {X 113.854,Y -41.308,Z -37.927,A -90.000,B 90.000,C 0.000} C_DIS
LIN {X 113.944,Y -41.308,Z -38.000,A -90.000,B 90.000,C 0.000} C_DIS
LIN {X 114.184,Y -41.308,Z -38.212,A -90.000,B 90.000,C 0.000} C_DIS
LIN {X 114.364,Y -41.308,Z -38.376,A -90.000,B 90.000,C 0.000} C_DIS
LIN {X 114.491,Y -41.308,Z -38.508,A -90.000,B 90.000,C 0.000} C_DIS
LIN {X 114.659,Y -41.308,Z -38.693,A -90.000,B 90.000,C 0.000} C_DIS
LIN {X 114.770,Y -41.308,Z -38.839,A -90.000,B 90.000,C 0.000} C_DIS
LIN {X 114.916,Y -41.308,Z -39.042,A -90.000,B 90.000,C 0.000} C_DIS
LIN {X 115.069,Y -41.308,Z -39.266,A -90.000,B 90.000,C 0.000} C_DIS
LIN {X 115.190,Y -41.308,Z -39.472,A -90.000,B 90.000,C 0.000} C_DIS
LIN {X 115.283,Y -41.308,Z -39.639,A -90.000,B 90.000,C 0.000} C_DIS
LIN {X 115.405,Y -41.308,Z -39.893,A -90.000,B 90.000,C 0.000} C_DIS
LIN {X 115.542,Y -41.308,Z -40.209,A -90.000,B 90.000,C 0.000} C_DIS
LIN {X 115.576,Y -41.308,Z -40.291,A -90.000,B 90.000,C 0.000} C_DIS
LIN {X 115.662,Y -41.308,Z -40.545,A -90.000,B 90.000,C 0.000} C_DIS
LIN {X 115.734,Y -41.308,Z -40.783,A -90.000,B 90.000,C 0.000} C_DIS
LIN {X 115.785,Y -41.308,Z -40.950,A -90.000,B 90.000,C 0.000} C_DIS
LIN {X 115.876,Y -41.308,Z -41.442,A -90.000,B 90.000,C 0.000} C_DIS
LIN {X 115.905,Y -41.308,Z -41.606,A -90.000,B 90.000,C 0.000} C_DIS
LIN {X 115.930,Y -41.308,Z -42.029,A -90.000,B 90.000,C 0.000} C_DIS
LIN {X 115.929,Y -41.308,Z -42.104,A -90.000,B 90.000,C 0.000} C_DIS
LIN {X 115.933,Y -41.308,Z -42.234,A -90.000,B 90.000,C 0.000} C_DIS
LIN {X 115.931,Y -41.308,Z -42.346,A -90.000,B 90.000,C 0.000} C_DIS
LIN {X 115.893,Y -41.308,Z -42.771,A -90.000,B 90.000,C 0.000} C_DIS
LIN {X 115.809,Y -41.308,Z -43.175,A -90.000,B 90.000,C 0.000} C_DIS
LIN {X 115.760,Y -41.308,Z -43.389,A -90.000,B 90.000,C 0.000} C_DIS
LIN {X 115.626,Y -41.308,Z -43.790,A -90.000,B 90.000,C 0.000} C_DIS
LIN {X 115.509,Y -41.308,Z -44.055,A -90.000,B 90.000,C 0.000} C_DIS
LIN {X 115.339,Y -41.308,Z -44.418,A -90.000,B 90.000,C 0.000} C_DIS
LIN {X 115.198,Y -41.308,Z -44.670,A -90.000,B 90.000,C 0.000} C_DIS
LIN {X 115.177,Y -41.308,Z -44.715,A -90.000,B 90.000,C 0.000} C_DIS
LIN {X 115.106,Y -41.308,Z -44.834,A -90.000,B 90.000,C 0.000} C_DIS
LIN {X 115.085,Y -41.308,Z -44.885,A -90.000,B 90.000,C 0.000} C_DIS
LIN {X 115.021,Y -41.308,Z -45.066,A -90.000,B 90.000,C 0.000} C_DIS
LIN {X 114.983,Y -41.308,Z -45.196,A -90.000,B 90.000,C 0.000} C_DIS
LIN {X 114.885,Y -41.308,Z -45.580,A -90.000,B 90.000,C 0.000} C_DIS
LIN {X 114.708,Y -41.308,Z -46.363,A -90.000,B 90.000,C 0.000} C_DIS
LIN {X 114.646,Y -41.308,Z -46.599,A -90.000,B 90.000,C 0.000} C_DIS
LIN {X 114.556,Y -41.308,Z -46.960,A -90.000,B 90.000,C 0.000} C_DIS
LIN {X 114.337,Y -41.308,Z -47.738,A -90.000,B 90.000,C 0.000} C_DIS
LIN {X 114.251,Y -41.308,Z -48.053,A -90.000,B 90.000,C 0.000} C_DIS
LIN {X 114.180,Y -41.308,Z -48.275,A -90.000,B 90.000,C 0.000} C_DIS
LIN {X 114.037,Y -41.308,Z -48.692,A -90.000,B 90.000,C 0.000} C_DIS
LIN {X 113.793,Y -41.308,Z -49.388,A -90.000,B 90.000,C 0.000} C_DIS
LIN {X 113.714,Y -41.308,Z -49.607,A -90.000,B 90.000,C 0.000} C_DIS
LIN {X 113.171,Y -41.308,Z -50.898,A -90.000,B 90.000,C 0.000} C_DIS
LIN {X 112.455,Y -41.308,Z -52.536,A -90.000,B 90.000,C 0.000} C_DIS
LIN {X 111.820,Y -41.308,Z -53.934,A -90.000,B 90.000,C 0.000} C_DIS
LIN {X 111.320,Y -41.308,Z -55.120,A -90.000,B 90.000,C 0.000} C_DIS
LIN {X 111.131,Y -41.308,Z -55.560,A -90.000,B 90.000,C 0.000} C_DIS
LIN {X 110.629,Y -41.308,Z -56.838,A -90.000,B 90.000,C 0.000} C_DIS
LIN {X 110.446,Y -41.308,Z -57.296,A -90.000,B 90.000,C 0.000} C_DIS
LIN {X 109.865,Y -41.308,Z -58.871,A -90.000,B 90.000,C 0.000} C_DIS
LIN {X 109.228,Y -41.308,Z -60.730,A -90.000,B 90.000,C 0.000} C_DIS
LIN {X 108.482,Y -41.308,Z -62.945,A -90.000,B 90.000,C 0.000} C_DIS
LIN {X 108.331,Y -41.308,Z -63.379,A -90.000,B 90.000,C 0.000} C_DIS
LIN {X 107.582,Y -41.308,Z -65.490,A -90.000,B 90.000,C 0.000} C_DIS
LIN {X 106.740,Y -41.308,Z -67.685,A -90.000,B 90.000,C 0.000} C_DIS
LIN {X 105.898,Y -41.308,Z -69.639,A -90.000,B 90.000,C 0.000} C_DIS
LIN {X 105.754,Y -41.308,Z -69.968,A -90.000,B 90.000,C 0.000} C_DIS
LIN {X 105.531,Y -41.308,Z -70.471,A -90.000,B 90.000,C 0.000} C_DIS
LIN {X 104.923,Y -41.308,Z -71.749,A -90.000,B 90.000,C 0.000} C_DIS
LIN {X 104.399,Y -41.308,Z -72.818,A -90.000,B 90.000,C 0.000} C_DIS
LIN {X 104.066,Y -41.308,Z -73.452,A -90.000,B 90.000,C 0.000} C_DIS
LIN {X 103.205,Y -41.308,Z -75.050,A -90.000,B 90.000,C 0.000} C_DIS
LIN {X 102.944,Y -41.308,Z -75.503,A -90.000,B 90.000,C 0.000} C_DIS
LIN {X 101.943,Y -41.308,Z -77.150,A -90.000,B 90.000,C 0.000} C_DIS
LIN {X 101.694,Y -41.308,Z -77.546,A -90.000,B 90.000,C 0.000} C_DIS
LIN {X 100.526,Y -41.308,Z -79.161,A -90.000,B 90.000,C 0.000} C_DIS
LIN {X 100.239,Y -41.308,Z -79.520,A -90.000,B 90.000,C 0.000} C_DIS
LIN {X 99.403,Y -41.308,Z -80.525,A -90.000,B 90.000,C 0.000} C_DIS
LIN {X 98.995,Y -41.308,Z -81.010,A -90.000,B 90.000,C 0.000} C_DIS
LIN {X 97.780,Y -41.308,Z -82.340,A -90.000,B 90.000,C 0.000} C_DIS
LIN {X 97.435,Y -41.308,Z -82.680,A -90.000,B 90.000,C 0.000} C_DIS
LIN {X 96.688,Y -41.308,Z -83.390,A -90.000,B 90.000,C 0.000} C_DIS
LIN {X 96.249,Y -41.308,Z -83.751,A -90.000,B 90.000,C 0.000} C_DIS
LIN {X 95.539,Y -41.308,Z -84.269,A -90.000,B 90.000,C 0.000} C_DIS
LIN {X 94.922,Y -41.308,Z -84.681,A -90.000,B 90.000,C 0.000} C_DIS
LIN {X 93.723,Y -41.308,Z -85.444,A -90.000,B 90.000,C 0.000} C_DIS
LIN {X 93.323,Y -41.308,Z -85.660,A -90.000,B 90.000,C 0.000} C_DIS
LIN {X 92.840,Y -41.308,Z -85.908,A -90.000,B 90.000,C 0.000} C_DIS
LIN {X 92.298,Y -41.308,Z -86.155,A -90.000,B 90.000,C 0.000} C_DIS
LIN {X 91.434,Y -41.308,Z -86.640,A -90.000,B 90.000,C 0.000} C_DIS
LIN {X 91.271,Y -41.308,Z -86.725,A -90.000,B 90.000,C 0.000} C_DIS
LIN {X 90.998,Y -41.308,Z -86.914,A -90.000,B 90.000,C 0.000} C_DIS
LIN {X 90.783,Y -41.308,Z -87.044,A -90.000,B 90.000,C 0.000} C_DIS
LIN {X 90.526,Y -41.308,Z -87.304,A -90.000,B 90.000,C 0.000} C_DIS
LIN {X 90.389,Y -41.308,Z -87.504,A -90.000,B 90.000,C 0.000} C_DIS
LIN {X 90.306,Y -41.308,Z -87.654,A -90.000,B 90.000,C 0.000} C_DIS
LIN {X 90.099,Y -41.308,Z -88.188,A -90.000,B 90.000,C 0.000} C_DIS
LIN {X 89.890,Y -41.308,Z -89.224,A -90.000,B 90.000,C 0.000} C_DIS
LIN {X 89.772,Y -41.308,Z -90.537,A -90.000,B 90.000,C 0.000} C_DIS
LIN {X 89.761,Y -41.308,Z -90.766,A -90.000,B 90.000,C 0.000} C_DIS
LIN {X 89.678,Y -41.308,Z -92.258,A -90.000,B 90.000,C 0.000} C_DIS
LIN {X 89.556,Y -41.308,Z -93.931,A -90.000,B 90.000,C 0.000} C_DIS
LIN {X 89.522,Y -41.308,Z -94.280,A -90.000,B 90.000,C 0.000} C_DIS
LIN {X 89.300,Y -41.308,Z -95.719,A -90.000,B 90.000,C 0.000} C_DIS
LIN {X 89.217,Y -41.308,Z -96.060,A -90.000,B 90.000,C 0.000} C_DIS
LIN {X 88.825,Y -41.308,Z -97.082,A -90.000,B 90.000,C 0.000} C_DIS
LIN {X 88.695,Y -41.308,Z -97.408,A -90.000,B 90.000,C 0.000} C_DIS
LIN {X 88.519,Y -41.308,Z -97.712,A -90.000,B 90.000,C 0.000} C_DIS
LIN {X 87.993,Y -41.308,Z -98.474,A -90.000,B 90.000,C 0.000} C_DIS
LIN {X 87.776,Y -41.308,Z -98.751,A -90.000,B 90.000,C 0.000} C_DIS
LIN {X 87.622,Y -41.308,Z -98.913,A -90.000,B 90.000,C 0.000} C_DIS
LIN {X 87.124,Y -41.308,Z -99.446,A -90.000,B 90.000,C 0.000} C_DIS
LIN {X 86.867,Y -41.308,Z -99.691,A -90.000,B 90.000,C 0.000} C_DIS
LIN {X 86.433,Y -41.308,Z -100.047,A -90.000,B 90.000,C 0.000} C_DIS
LIN {X 85.899,Y -41.308,Z -100.605,A -90.000,B 90.000,C 0.000} C_DIS
LIN {X 85.811,Y -41.308,Z -100.699,A -90.000,B 90.000,C 0.000} C_DIS
LIN {X 85.470,Y -41.308,Z -101.163,A -90.000,B 90.000,C 0.000} C_DIS
LIN {X 85.206,Y -41.308,Z -101.528,A -90.000,B 90.000,C 0.000} C_DIS
LIN {X 85.091,Y -41.308,Z -101.750,A -90.000,B 90.000,C 0.000} C_DIS
LIN {X 84.773,Y -41.308,Z -102.347,A -90.000,B 90.000,C 0.000} C_DIS
LIN {X 84.752,Y -41.308,Z -102.429,A -90.000,B 90.000,C 0.000} C_DIS
LIN {X 84.572,Y -41.308,Z -103.024,A -90.000,B 90.000,C 0.000} C_DIS
LIN {X 84.573,Y -41.308,Z -103.637,A -90.000,B 90.000,C 0.000} C_DIS
LIN {X 84.677,Y -41.308,Z -104.414,A -90.000,B 90.000,C 0.000} C_DIS
LIN {X 84.758,Y -41.308,Z -104.751,A -90.000,B 90.000,C 0.000} C_DIS
LIN {X 84.829,Y -41.308,Z -105.567,A -90.000,B 90.000,C 0.000} C_DIS
LIN {X 84.977,Y -41.308,Z -106.244,A -90.000,B 90.000,C 0.000} C_DIS
LIN {X 85.002,Y -41.308,Z -106.525,A -90.000,B 90.000,C 0.000} C_DIS
LIN {X 84.997,Y -41.308,Z -106.654,A -90.000,B 90.000,C 0.000} C_DIS
LIN {X 84.956,Y -41.308,Z -107.107,A -90.000,B 90.000,C 0.000} C_DIS
LIN {X 84.991,Y -41.308,Z -108.122,A -90.000,B 90.000,C 0.000} C_DIS
LIN {X 84.985,Y -41.308,Z -108.251,A -90.000,B 90.000,C 0.000} C_DIS
LIN {X 84.938,Y -41.308,Z -108.529,A -90.000,B 90.000,C 0.000} C_DIS
LIN {X 84.704,Y -41.308,Z -109.209,A -90.000,B 90.000,C 0.000} C_DIS
LIN {X 84.387,Y -41.308,Z -110.494,A -90.000,B 90.000,C 0.000} C_DIS
LIN {X 84.292,Y -41.308,Z -110.759,A -90.000,B 90.000,C 0.000} C_DIS
LIN {X 83.759,Y -41.308,Z -111.966,A -90.000,B 90.000,C 0.000} C_DIS
LIN {X 83.377,Y -41.308,Z -112.997,A -90.000,B 90.000,C 0.000} C_DIS
LIN {X 82.675,Y -41.308,Z -114.644,A -90.000,B 90.000,C 0.000} C_DIS
LIN {X 82.475,Y -41.308,Z -115.169,A -90.000,B 90.000,C 0.000} C_DIS
LIN {X 81.908,Y -41.308,Z -117.104,A -90.000,B 90.000,C 0.000} C_DIS
LIN {X 81.847,Y -41.308,Z -117.319,A -90.000,B 90.000,C 0.000} C_DIS
LIN {X 81.837,Y -41.308,Z -117.488,A -90.000,B 90.000,C 0.000} C_DIS
LIN {X 81.823,Y -41.308,Z -119.354,A -90.000,B 90.000,C 0.000} C_DIS
LIN {X 82.180,Y -41.308,Z -121.212,A -90.000,B 90.000,C 0.000} C_DIS
LIN {X 82.207,Y -41.308,Z -121.372,A -90.000,B 90.000,C 0.000} C_DIS
LIN {X 82.651,Y -41.308,Z -122.944,A -90.000,B 90.000,C 0.000} C_DIS
LIN {X 82.723,Y -41.308,Z -123.210,A -90.000,B 90.000,C 0.000} C_DIS
LIN {X 82.779,Y -41.308,Z -123.598,A -90.000,B 90.000,C 0.000} C_DIS
LIN {X 83.173,Y -41.308,Z -125.135,A -90.000,B 90.000,C 0.000} C_DIS
LIN {X 83.331,Y -41.308,Z -126.417,A -90.000,B 90.000,C 0.000} C_DIS
LIN {X 83.356,Y -41.308,Z -126.698,A -90.000,B 90.000,C 0.000} C_DIS
LIN {X 83.405,Y -41.308,Z -128.592,A -90.000,B 90.000,C 0.000} C_DIS
LIN {X 83.374,Y -41.308,Z -129.313,A -90.000,B 90.000,C 0.000} C_DIS
LIN {X 83.344,Y -41.308,Z -130.665,A -90.000,B 90.000,C 0.000} C_DIS
LIN {X 83.338,Y -41.308,Z -130.793,A -90.000,B 90.000,C 0.000} C_DIS
LIN {X 83.281,Y -41.308,Z -131.583,A -90.000,B 90.000,C 0.000} C_DIS
LIN {X 83.238,Y -41.308,Z -133.072,A -90.000,B 90.000,C 0.000} C_DIS
LIN {X 83.222,Y -41.308,Z -133.321,A -90.000,B 90.000,C 0.000} C_DIS
LIN {X 83.170,Y -41.308,Z -134.097,A -90.000,B 90.000,C 0.000} C_DIS
LIN {X 83.137,Y -41.308,Z -134.907,A -90.000,B 90.000,C 0.000} C_DIS
LIN {X 83.115,Y -41.308,Z -137.034,A -90.000,B 90.000,C 0.000} C_DIS
LIN {X 83.072,Y -41.308,Z -138.244,A -90.000,B 90.000,C 0.000} C_DIS
LIN {X 83.050,Y -41.308,Z -140.397,A -90.000,B 90.000,C 0.000} C_DIS
LIN {X 82.979,Y -41.308,Z -142.045,A -90.000,B 90.000,C 0.000} C_DIS
LIN {X 82.934,Y -41.308,Z -144.011,A -90.000,B 90.000,C 0.000} C_DIS
LIN {X 82.802,Y -41.308,Z -146.158,A -90.000,B 90.000,C 0.000} C_DIS
LIN {X 82.727,Y -41.308,Z -147.785,A -90.000,B 90.000,C 0.000} C_DIS
LIN {X 82.488,Y -41.308,Z -150.423,A -90.000,B 90.000,C 0.000} C_DIS
LIN {X 82.394,Y -41.308,Z -151.605,A -90.000,B 90.000,C 0.000} C_DIS
LIN {X 82.361,Y -41.308,Z -151.923,A -90.000,B 90.000,C 0.000} C_DIS
LIN {X 81.975,Y -41.308,Z -154.987,A -90.000,B 90.000,C 0.000} C_DIS
LIN {X 81.887,Y -41.308,Z -155.731,A -90.000,B 90.000,C 0.000} C_DIS
LIN {X 81.326,Y -41.308,Z -159.059,A -90.000,B 90.000,C 0.000} C_DIS
LIN {X 81.257,Y -41.308,Z -159.478,A -90.000,B 90.000,C 0.000} C_DIS
LIN {X 80.448,Y -41.308,Z -163.143,A -90.000,B 90.000,C 0.000} C_DIS
LIN {X 80.372,Y -41.308,Z -163.430,A -90.000,B 90.000,C 0.000} C_DIS
LIN {X 79.377,Y -41.308,Z -166.927,A -90.000,B 90.000,C 0.000} C_DIS
LIN {X 78.292,Y -41.308,Z -170.276,A -90.000,B 90.000,C 0.000} C_DIS
LIN {X 77.217,Y -41.308,Z -173.471,A -90.000,B 90.000,C 0.000} C_DIS
LIN {X 76.261,Y -41.308,Z -176.488,A -90.000,B 90.000,C 0.000} C_DIS
LIN {X 75.722,Y -41.308,Z -178.546,A -90.000,B 90.000,C 0.000} C_DIS
LIN {X 75.582,Y -41.308,Z -179.099,A -90.000,B 90.000,C 0.000} C_DIS
LIN {X 75.046,Y -41.308,Z -181.535,A -90.000,B 90.000,C 0.000} C_DIS
LIN {X 74.977,Y -41.308,Z -181.866,A -90.000,B 90.000,C 0.000} C_DIS
LIN {X 74.459,Y -41.308,Z -184.522,A -90.000,B 90.000,C 0.000} C_DIS
LIN {X 74.391,Y -41.308,Z -184.883,A -90.000,B 90.000,C 0.000} C_DIS
LIN {X 73.952,Y -41.308,Z -187.066,A -90.000,B 90.000,C 0.000} C_DIS
LIN {X 73.636,Y -41.308,Z -188.548,A -90.000,B 90.000,C 0.000} C_DIS
LIN {X 73.397,Y -41.308,Z -189.565,A -90.000,B 90.000,C 0.000} C_DIS
LIN {X 73.331,Y -41.308,Z -189.831,A -90.000,B 90.000,C 0.000} C_DIS
LIN {X 72.687,Y -41.308,Z -192.299,A -90.000,B 90.000,C 0.000} C_DIS
LIN {X 72.046,Y -41.308,Z -194.469,A -90.000,B 90.000,C 0.000} C_DIS
LIN {X 71.753,Y -41.308,Z -195.437,A -90.000,B 90.000,C 0.000} C_DIS
LIN {X 70.653,Y -41.308,Z -198.705,A -90.000,B 90.000,C 0.000} C_DIS
LIN {X 70.547,Y -41.308,Z -198.992,A -90.000,B 90.000,C 0.000} C_DIS
LIN {X 69.234,Y -41.308,Z -202.588,A -90.000,B 90.000,C 0.000} C_DIS
LIN {X 69.034,Y -41.308,Z -203.100,A -90.000,B 90.000,C 0.000} C_DIS
LIN {X 67.537,Y -41.308,Z -206.968,A -90.000,B 90.000,C 0.000} C_DIS
LIN {X 67.234,Y -41.308,Z -207.710,A -90.000,B 90.000,C 0.000} C_DIS
LIN {X 65.602,Y -41.308,Z -211.729,A -90.000,B 90.000,C 0.000} C_DIS
LIN {X 65.186,Y -41.308,Z -212.706,A -90.000,B 90.000,C 0.000} C_DIS
LIN {X 63.468,Y -41.308,Z -216.755,A -90.000,B 90.000,C 0.000} C_DIS
LIN {X 61.631,Y -41.308,Z -220.908,A -90.000,B 90.000,C 0.000} C_DIS
LIN {X 61.011,Y -41.308,Z -222.298,A -90.000,B 90.000,C 0.000} C_DIS
LIN {X 58.767,Y -41.308,Z -227.036,A -90.000,B 90.000,C 0.000} C_DIS
LIN {X 58.529,Y -41.308,Z -227.542,A -90.000,B 90.000,C 0.000} C_DIS
LIN {X 56.687,Y -41.308,Z -231.093,A -90.000,B 90.000,C 0.000} C_DIS
LIN {X 55.799,Y -41.308,Z -232.848,A -90.000,B 90.000,C 0.000} C_DIS
LIN {X 53.764,Y -41.308,Z -236.369,A -90.000,B 90.000,C 0.000} C_DIS
LIN {X 52.792,Y -41.308,Z -238.142,A -90.000,B 90.000,C 0.000} C_DIS
LIN {X 51.738,Y -41.308,Z -239.895,A -90.000,B 90.000,C 0.000} C_DIS
LIN {X 51.546,Y -41.308,Z -240.211,A -90.000,B 90.000,C 0.000} C_DIS
LIN {X 49.336,Y -41.308,Z -243.561,A -90.000,B 90.000,C 0.000} C_DIS
LIN {X 49.336,Y -60.000,Z -243.561,A -90.000,B 90.000,C 0.000} C_DIS
LIN {X 26.911,Y -60.000,Z -77.635,A -90.000,B 90.000,C 0.000} C_DIS
LIN {X 26.911,Y -41.308,Z -77.635,A -90.000,B 90.000,C 0.000} C_DIS
LIN {X 26.895,Y -41.308,Z -77.635,A -90.000,B 90.000,C 0.000} C_DIS
LIN {X 25.157,Y -41.308,Z -77.463,A -90.000,B 90.000,C 0.000} C_DIS
LIN {X 24.968,Y -41.308,Z -77.429,A -90.000,B 90.000,C 0.000} C_DIS
LIN {X 24.759,Y -41.308,Z -77.343,A -90.000,B 90.000,C 0.000} C_DIS
LIN {X 23.229,Y -41.308,Z -76.469,A -90.000,B 90.000,C 0.000} C_DIS
LIN {X 23.138,Y -41.308,Z -76.407,A -90.000,B 90.000,C 0.000} C_DIS
LIN {X 23.064,Y -41.308,Z -76.347,A -90.000,B 90.000,C 0.000} C_DIS
LIN {X 22.987,Y -41.308,Z -76.267,A -90.000,B 90.000,C 0.000} C_DIS
LIN {X 22.932,Y -41.308,Z -76.189,A -90.000,B 90.000,C 0.000} C_DIS
LIN {X 22.642,Y -41.308,Z -75.749,A -90.000,B 90.000,C 0.000} C_DIS
LIN {X 22.583,Y -41.308,Z -75.579,A -90.000,B 90.000,C 0.000} C_DIS
LIN {X 22.572,Y -41.308,Z -75.400,A -90.000,B 90.000,C 0.000} C_DIS
LIN {X 22.611,Y -41.308,Z -75.225,A -90.000,B 90.000,C 0.000} C_DIS
LIN {X 22.638,Y -41.308,Z -75.147,A -90.000,B 90.000,C 0.000} C_DIS
LIN {X 22.689,Y -41.308,Z -75.074,A -90.000,B 90.000,C 0.000} C_DIS
LIN {X 22.822,Y -41.308,Z -74.940,A -90.000,B 90.000,C 0.000} C_DIS
LIN {X 22.978,Y -41.308,Z -74.851,A -90.000,B 90.000,C 0.000} C_DIS
LIN {X 23.152,Y -41.308,Z -74.809,A -90.000,B 90.000,C 0.000} C_DIS
LIN {X 23.337,Y -41.308,Z -74.801,A -90.000,B 90.000,C 0.000} C_DIS
LIN {X 23.765,Y -41.308,Z -74.723,A -90.000,B 90.000,C 0.000} C_DIS
LIN {X 23.944,Y -41.308,Z -74.731,A -90.000,B 90.000,C 0.000} C_DIS
LIN {X 24.474,Y -41.308,Z -74.880,A -90.000,B 90.000,C 0.000} C_DIS
LIN {X 24.644,Y -41.308,Z -74.936,A -90.000,B 90.000,C 0.000} C_DIS
LIN {X 25.713,Y -41.308,Z -75.312,A -90.000,B 90.000,C 0.000} C_DIS
LIN {X 25.763,Y -41.308,Z -75.334,A -90.000,B 90.000,C 0.000} C_DIS
LIN {X 26.089,Y -41.308,Z -75.549,A -90.000,B 90.000,C 0.000} C_DIS
LIN {X 26.237,Y -41.308,Z -75.650,A -90.000,B 90.000,C 0.000} C_DIS
LIN {X 26.588,Y -41.308,Z -75.968,A -90.000,B 90.000,C 0.000} C_DIS
LIN {X 27.184,Y -41.308,Z -76.338,A -90.000,B 90.000,C 0.000} C_DIS
LIN {X 27.332,Y -41.308,Z -76.439,A -90.000,B 90.000,C 0.000} C_DIS
LIN {X 27.357,Y -41.308,Z -76.462,A -90.000,B 90.000,C 0.000} C_DIS
LIN {X 27.401,Y -41.308,Z -76.494,A -90.000,B 90.000,C 0.000} C_DIS
LIN {X 27.511,Y -41.308,Z -76.625,A -90.000,B 90.000,C 0.000} C_DIS
LIN {X 27.516,Y -41.308,Z -76.632,A -90.000,B 90.000,C 0.000} C_DIS
LIN {X 27.589,Y -41.308,Z -76.795,A -90.000,B 90.000,C 0.000} C_DIS
LIN {X 27.659,Y -41.308,Z -77.082,A -90.000,B 90.000,C 0.000} C_DIS
LIN {X 27.657,Y -41.308,Z -77.101,A -90.000,B 90.000,C 0.000} C_DIS
LIN {X 27.623,Y -41.308,Z -77.183,A -90.000,B 90.000,C 0.000} C_DIS
LIN {X 27.455,Y -41.308,Z -77.398,A -90.000,B 90.000,C 0.000} C_DIS
LIN {X 27.320,Y -41.308,Z -77.515,A -90.000,B 90.000,C 0.000} C_DIS
LIN {X 27.157,Y -41.308,Z -77.591,A -90.000,B 90.000,C 0.000} C_DIS
LIN {X 27.076,Y -41.308,Z -77.608,A -90.000,B 90.000,C 0.000} C_DIS
LIN {X 26.911,Y -41.308,Z -77.635,A -90.000,B 90.000,C 0.000} C_DIS
LIN {X 26.911,Y -60.000,Z -77.635,A -90.000,B 90.000,C 0.000} C_DIS
LIN {X 59.784,Y -60.000,Z -109.242,A -90.000,B 90.000,C 0.000} C_DIS
LIN {X 59.784,Y -39.308,Z -109.242,A -90.000,B 90.000,C 0.000} C_DIS
LIN {X 58.768,Y -39.308,Z -111.415,A -90.000,B 90.000,C 0.000} C_DIS
LIN {X 58.532,Y -39.308,Z -112.196,A -90.000,B 90.000,C 0.000} C_DIS
LIN {X 58.530,Y -39.308,Z -112.201,A -90.000,B 90.000,C 0.000} C_DIS
LIN {X 58.531,Y -39.308,Z -112.502,A -90.000,B 90.000,C 0.000} C_DIS
LIN {X 58.496,Y -39.308,Z -112.765,A -90.000,B 90.000,C 0.000} C_DIS
LIN {X 59.222,Y -39.308,Z -111.842,A -90.000,B 90.000,C 0.000} C_DIS
LIN {X 59.906,Y -39.308,Z -109.794,A -90.000,B 90.000,C 0.000} C_DIS
LIN {X 60.094,Y -39.308,Z -109.174,A -90.000,B 90.000,C 0.000} C_DIS
LIN {X 59.784,Y -39.308,Z -109.242,A -90.000,B 90.000,C 0.000} C_DIS
LIN {X 59.784,Y -60.000,Z -109.242,A -90.000,B 90.000,C 0.000} C_DIS
LIN {X -80.206,Y -60.000,Z -243.561,A -90.000,B 90.000,C 0.000} C_DIS
LIN {X -80.206,Y -40.663,Z -243.561,A -90.000,B 90.000,C 0.000} C_DIS
LIN {X -80.202,Y -40.649,Z -243.535,A -90.000,B 90.000,C 0.000} C_DIS
LIN {X -80.143,Y -40.540,Z -243.312,A -90.000,B 90.000,C 0.000} C_DIS
LIN {X -80.092,Y -40.478,Z -243.178,A -90.000,B 90.000,C 0.000} C_DIS
LIN {X -80.055,Y -40.443,Z -243.095,A -90.000,B 90.000,C 0.000} C_DIS
LIN {X -79.985,Y -40.389,Z -242.963,A -90.000,B 90.000,C 0.000} C_DIS
LIN {X -79.816,Y -40.299,Z -242.711,A -90.000,B 90.000,C 0.000} C_DIS
LIN {X -79.640,Y -40.242,Z -242.511,A -90.000,B 90.000,C 0.000} C_DIS
LIN {X -79.602,Y -40.233,Z -242.473,A -90.000,B 90.000,C 0.000} C_DIS
LIN {X -79.147,Y -40.187,Z -242.130,A -90.000,B 90.000,C 0.000} C_DIS
LIN {X -77.511,Y -40.188,Z -241.177,A -90.000,B 90.000,C 0.000} C_DIS
LIN {X -74.607,Y -40.211,Z -239.526,A -90.000,B 90.000,C 0.000} C_DIS
LIN {X -72.699,Y -40.211,Z -238.453,A -90.000,B 90.000,C 0.000} C_DIS
LIN {X -71.839,Y -40.204,Z -237.974,A -90.000,B 90.000,C 0.000} C_DIS
LIN {X -71.481,Y -40.203,Z -237.778,A -90.000,B 90.000,C 0.000} C_DIS
LIN {X -68.474,Y -40.218,Z -236.172,A -90.000,B 90.000,C 0.000} C_DIS
LIN {X -63.905,Y -40.218,Z -233.750,A -90.000,B 90.000,C 0.000} C_DIS
LIN {X -62.954,Y -40.209,Z -233.252,A -90.000,B 90.000,C 0.000} C_DIS
LIN {X -59.110,Y -40.208,Z -231.296,A -90.000,B 90.000,C 0.000} C_DIS
LIN {X -56.183,Y -40.219,Z -229.825,A -90.000,B 90.000,C 0.000} C_DIS
LIN {X -54.737,Y -40.217,Z -229.103,A -90.000,B 90.000,C 0.000} C_DIS
LIN {X -53.328,Y -40.217,Z -228.405,A -90.000,B 90.000,C 0.000} C_DIS
LIN {X -51.128,Y -40.223,Z -227.328,A -90.000,B 90.000,C 0.000} C_DIS
LIN {X -50.446,Y -40.227,Z -226.999,A -90.000,B 90.000,C 0.000} C_DIS
LIN {X -47.677,Y -40.236,Z -225.664,A -90.000,B 90.000,C 0.000} C_DIS
LIN {X -45.969,Y -40.253,Z -224.860,A -90.000,B 90.000,C 0.000} C_DIS
LIN {X -44.872,Y -40.260,Z -224.337,A -90.000,B 90.000,C 0.000} C_DIS
LIN {X -42.330,Y -40.273,Z -223.127,A -90.000,B 90.000,C 0.000} C_DIS
LIN {X -40.892,Y -40.288,Z -222.458,A -90.000,B 90.000,C 0.000} C_DIS
LIN {X -39.657,Y -40.295,Z -221.887,A -90.000,B 90.000,C 0.000} C_DIS
LIN {X -39.010,Y -40.295,Z -221.591,A -90.000,B 90.000,C 0.000} C_DIS
LIN {X -37.991,Y -40.303,Z -221.119,A -90.000,B 90.000,C 0.000} C_DIS
LIN {X -37.270,Y -40.303,Z -220.776,A -90.000,B 90.000,C 0.000} C_DIS
LIN {X -35.889,Y -40.307,Z -220.127,A -90.000,B 90.000,C 0.000} C_DIS
LIN {X -34.884,Y -40.316,Z -219.665,A -90.000,B 90.000,C 0.000} C_DIS
LIN {X -33.878,Y -40.322,Z -219.206,A -90.000,B 90.000,C 0.000} C_DIS
LIN {X -32.033,Y -40.342,Z -218.379,A -90.000,B 90.000,C 0.000} C_DIS
LIN {X -31.717,Y -40.347,Z -218.241,A -90.000,B 90.000,C 0.000} C_DIS
LIN {X -30.961,Y -40.368,Z -217.906,A -90.000,B 90.000,C 0.000} C_DIS
LIN {X -27.871,Y -40.408,Z -216.435,A -90.000,B 90.000,C 0.000} C_DIS
LIN {X -27.196,Y -40.414,Z -216.114,A -90.000,B 90.000,C 0.000} C_DIS
LIN {X -25.802,Y -40.424,Z -215.451,A -90.000,B 90.000,C 0.000} C_DIS
LIN {X -24.739,Y -40.439,Z -214.941,A -90.000,B 90.000,C 0.000} C_DIS
LIN {X -23.924,Y -40.439,Z -214.524,A -90.000,B 90.000,C 0.000} C_DIS
LIN {X -21.928,Y -40.429,Z -213.476,A -90.000,B 90.000,C 0.000} C_DIS
LIN {X -20.405,Y -40.453,Z -212.728,A -90.000,B 90.000,C 0.000} C_DIS
LIN {X -19.962,Y -40.466,Z -212.507,A -90.000,B 90.000,C 0.000} C_DIS
LIN {X -19.642,Y -40.477,Z -212.352,A -90.000,B 90.000,C 0.000} C_DIS
LIN {X -18.577,Y -40.490,Z -211.777,A -90.000,B 90.000,C 0.000} C_DIS
LIN {X -16.600,Y -40.530,Z -210.701,A -90.000,B 90.000,C 0.000} C_DIS
LIN {X -15.817,Y -40.539,Z -210.257,A -90.000,B 90.000,C 0.000} C_DIS
LIN {X -15.697,Y -40.541,Z -210.189,A -90.000,B 90.000,C 0.000} C_DIS
LIN {X -15.042,Y -40.560,Z -209.811,A -90.000,B 90.000,C 0.000} C_DIS
LIN {X -14.540,Y -40.570,Z -209.506,A -90.000,B 90.000,C 0.000} C_DIS
LIN {X -13.438,Y -40.575,Z -208.840,A -90.000,B 90.000,C 0.000} C_DIS
LIN {X -12.255,Y -40.571,Z -208.096,A -90.000,B 90.000,C 0.000} C_DIS
LIN {X -11.766,Y -40.567,Z -207.789,A -90.000,B 90.000,C 0.000} C_DIS
LIN {X -10.811,Y -40.575,Z -207.183,A -90.000,B 90.000,C 0.000} C_DIS
LIN {X -8.729,Y -40.569,Z -205.788,A -90.000,B 90.000,C 0.000} C_DIS
LIN {X -8.657,Y -40.569,Z -205.741,A -90.000,B 90.000,C 0.000} C_DIS
LIN {X -7.526,Y -40.587,Z -205.048,A -90.000,B 90.000,C 0.000} C_DIS
LIN {X -6.627,Y -40.619,Z -204.488,A -90.000,B 90.000,C 0.000} C_DIS
LIN {X -5.390,Y -40.625,Z -203.603,A -90.000,B 90.000,C 0.000} C_DIS
LIN {X -3.614,Y -40.645,Z -202.379,A -90.000,B 90.000,C 0.000} C_DIS
LIN {X -2.810,Y -40.671,Z -201.818,A -90.000,B 90.000,C 0.000} C_DIS
LIN {X -0.183,Y -40.662,Z -199.664,A -90.000,B 90.000,C 0.000} C_DIS
LIN {X 0.104,Y -40.662,Z -199.439,A -90.000,B 90.000,C 0.000} C_DIS
LIN {X 0.741,Y -40.682,Z -198.935,A -90.000,B 90.000,C 0.000} C_DIS
LIN {X 3.647,Y -40.638,Z -196.190,A -90.000,B 90.000,C 0.000} C_DIS
LIN {X 3.937,Y -40.641,Z -195.913,A -90.000,B 90.000,C 0.000} C_DIS
LIN {X 4.185,Y -40.647,Z -195.687,A -90.000,B 90.000,C 0.000} C_DIS
LIN {X 4.232,Y -40.647,Z -195.640,A -90.000,B 90.000,C 0.000} C_DIS
LIN {X 6.673,Y -40.593,Z -192.986,A -90.000,B 90.000,C 0.000} C_DIS
LIN {X 7.195,Y -40.590,Z -192.413,A -90.000,B 90.000,C 0.000} C_DIS
LIN {X 7.299,Y -40.590,Z -192.301,A -90.000,B 90.000,C 0.000} C_DIS
LIN {X 9.817,Y -40.531,Z -189.387,A -90.000,B 90.000,C 0.000} C_DIS
LIN {X 10.165,Y -40.530,Z -188.980,A -90.000,B 90.000,C 0.000} C_DIS
LIN {X 12.623,Y -40.470,Z -186.098,A -90.000,B 90.000,C 0.000} C_DIS
LIN {X 13.105,Y -40.467,Z -185.527,A -90.000,B 90.000,C 0.000} C_DIS
LIN {X 13.224,Y -40.462,Z -185.384,A -90.000,B 90.000,C 0.000} C_DIS
LIN {X 15.662,Y -40.409,Z -182.637,A -90.000,B 90.000,C 0.000} C_DIS
LIN {X 15.845,Y -40.409,Z -182.428,A -90.000,B 90.000,C 0.000} C_DIS
LIN {X 15.948,Y -40.404,Z -182.308,A -90.000,B 90.000,C 0.000} C_DIS
LIN {X 16.165,Y -40.393,Z -182.066,A -90.000,B 90.000,C 0.000} C_DIS
LIN {X 16.276,Y -40.390,Z -181.948,A -90.000,B 90.000,C 0.000} C_DIS
LIN {X 18.230,Y -40.361,Z -179.957,A -90.000,B 90.000,C 0.000} C_DIS
LIN {X 18.724,Y -40.353,Z -179.456,A -90.000,B 90.000,C 0.000} C_DIS
LIN {X 18.992,Y -40.349,Z -179.189,A -90.000,B 90.000,C 0.000} C_DIS
LIN {X 19.311,Y -40.349,Z -178.881,A -90.000,B 90.000,C 0.000} C_DIS
LIN {X 21.014,Y -40.335,Z -177.255,A -90.000,B 90.000,C 0.000} C_DIS
LIN {X 21.631,Y -40.328,Z -176.657,A -90.000,B 90.000,C 0.000} C_DIS
LIN {X 22.562,Y -40.315,Z -175.763,A -90.000,B 90.000,C 0.000} C_DIS
LIN {X 22.796,Y -40.314,Z -175.543,A -90.000,B 90.000,C 0.000} C_DIS
LIN {X 23.136,Y -40.318,Z -175.218,A -90.000,B 90.000,C 0.000} C_DIS
LIN {X 24.416,Y -40.303,Z -173.927,A -90.000,B 90.000,C 0.000} C_DIS
LIN {X 24.799,Y -40.312,Z -173.529,A -90.000,B 90.000,C 0.000} C_DIS
LIN {X 25.033,Y -40.310,Z -173.265,A -90.000,B 90.000,C 0.000} C_DIS
LIN {X 26.087,Y -40.292,Z -172.059,A -90.000,B 90.000,C 0.000} C_DIS
LIN {X 26.335,Y -40.297,Z -171.767,A -90.000,B 90.000,C 0.000} C_DIS
LIN {X 26.680,Y -40.288,Z -171.320,A -90.000,B 90.000,C 0.000} C_DIS
LIN {X 27.187,Y -40.280,Z -170.675,A -90.000,B 90.000,C 0.000} C_DIS
LIN {X 27.516,Y -40.274,Z -170.257,A -90.000,B 90.000,C 0.000} C_DIS
LIN {X 27.655,Y -40.274,Z -170.078,A -90.000,B 90.000,C 0.000} C_DIS
LIN {X 28.253,Y -40.257,Z -169.223,A -90.000,B 90.000,C 0.000} C_DIS
LIN {X 28.863,Y -40.245,Z -168.373,A -90.000,B 90.000,C 0.000} C_DIS
LIN {X 29.044,Y -40.246,Z -168.117,A -90.000,B 90.000,C 0.000} C_DIS
LIN {X 29.953,Y -40.221,Z -166.725,A -90.000,B 90.000,C 0.000} C_DIS
LIN {X 30.268,Y -40.216,Z -166.253,A -90.000,B 90.000,C 0.000} C_DIS
LIN {X 30.358,Y -40.217,Z -166.115,A -90.000,B 90.000,C 0.000} C_DIS
LIN {X 30.584,Y -40.207,Z -165.742,A -90.000,B 90.000,C 0.000} C_DIS
LIN {X 31.656,Y -40.173,Z -164.004,A -90.000,B 90.000,C 0.000} C_DIS
LIN {X 31.801,Y -40.173,Z -163.764,A -90.000,B 90.000,C 0.000} C_DIS
LIN {X 32.397,Y -40.149,Z -162.726,A -90.000,B 90.000,C 0.000} C_DIS
LIN {X 32.937,Y -40.132,Z -161.798,A -90.000,B 90.000,C 0.000} C_DIS
LIN {X 33.230,Y -40.133,Z -161.280,A -90.000,B 90.000,C 0.000} C_DIS
LIN {X 33.989,Y -40.113,Z -159.860,A -90.000,B 90.000,C 0.000} C_DIS
LIN {X 34.589,Y -40.123,Z -158.703,A -90.000,B 90.000,C 0.000} C_DIS
LIN {X 34.984,Y -40.117,Z -157.899,A -90.000,B 90.000,C 0.000} C_DIS
LIN {X 35.398,Y -40.133,Z -157.020,A -90.000,B 90.000,C 0.000} C_DIS
LIN {X 35.736,Y -40.151,Z -156.294,A -90.000,B 90.000,C 0.000} C_DIS
LIN {X 35.952,Y -40.153,Z -155.803,A -90.000,B 90.000,C 0.000} C_DIS
LIN {X 36.302,Y -40.190,Z -154.947,A -90.000,B 90.000,C 0.000} C_DIS
LIN {X 36.825,Y -40.225,Z -153.769,A -90.000,B 90.000,C 0.000} C_DIS
LIN {X 36.866,Y -40.227,Z -153.671,A -90.000,B 90.000,C 0.000} C_DIS
LIN {X 36.939,Y -40.237,Z -153.475,A -90.000,B 90.000,C 0.000} C_DIS
LIN {X 37.042,Y -40.253,Z -153.195,A -90.000,B 90.000,C 0.000} C_DIS
LIN {X 37.350,Y -40.267,Z -152.413,A -90.000,B 90.000,C 0.000} C_DIS
LIN {X 37.416,Y -40.272,Z -152.257,A -90.000,B 90.000,C 0.000} C_DIS
LIN {X 37.592,Y -40.295,Z -151.838,A -90.000,B 90.000,C 0.000} C_DIS
LIN {X 37.657,Y -40.302,Z -151.683,A -90.000,B 90.000,C 0.000} C_DIS
LIN {X 37.872,Y -40.314,Z -151.195,A -90.000,B 90.000,C 0.000} C_DIS
LIN {X 38.113,Y -40.341,Z -150.524,A -90.000,B 90.000,C 0.000} C_DIS
LIN {X 38.155,Y -40.347,Z -150.417,A -90.000,B 90.000,C 0.000} C_DIS
LIN {X 38.396,Y -40.386,Z -149.843,A -90.000,B 90.000,C 0.000} C_DIS
LIN {X 38.898,Y -40.401,Z -148.732,A -90.000,B 90.000,C 0.000} C_DIS
LIN {X 39.026,Y -40.422,Z -148.424,A -90.000,B 90.000,C 0.000} C_DIS
LIN {X 39.065,Y -40.428,Z -148.336,A -90.000,B 90.000,C 0.000} C_DIS
LIN {X 39.140,Y -40.440,Z -148.147,A -90.000,B 90.000,C 0.000} C_DIS
LIN {X 39.202,Y -40.450,Z -148.007,A -90.000,B 90.000,C 0.000} C_DIS
LIN {X 39.285,Y -40.454,Z -147.834,A -90.000,B 90.000,C 0.000} C_DIS
LIN {X 39.466,Y -40.458,Z -147.465,A -90.000,B 90.000,C 0.000} C_DIS
LIN {X 39.863,Y -40.456,Z -146.611,A -90.000,B 90.000,C 0.000} C_DIS
LIN {X 39.923,Y -40.460,Z -146.480,A -90.000,B 90.000,C 0.000} C_DIS
LIN {X 40.108,Y -40.474,Z -146.085,A -90.000,B 90.000,C 0.000} C_DIS
LIN {X 40.248,Y -40.486,Z -145.826,A -90.000,B 90.000,C 0.000} C_DIS
LIN {X 40.525,Y -40.486,Z -145.336,A -90.000,B 90.000,C 0.000} C_DIS
LIN {X 40.601,Y -40.483,Z -145.187,A -90.000,B 90.000,C 0.000} C_DIS
LIN {X 41.051,Y -40.503,Z -144.281,A -90.000,B 90.000,C 0.000} C_DIS
LIN {X 41.132,Y -40.507,Z -144.117,A -90.000,B 90.000,C 0.000} C_DIS
LIN {X 41.172,Y -40.509,Z -144.042,A -90.000,B 90.000,C 0.000} C_DIS
LIN {X 41.270,Y -40.518,Z -143.876,A -90.000,B 90.000,C 0.000} C_DIS
LIN {X 41.353,Y -40.518,Z -143.743,A -90.000,B 90.000,C 0.000} C_DIS
LIN {X 42.351,Y -40.510,Z -142.212,A -90.000,B 90.000,C 0.000} C_DIS
LIN {X 42.588,Y -40.516,Z -141.824,A -90.000,B 90.000,C 0.000} C_DIS
LIN {X 42.689,Y -40.516,Z -141.663,A -90.000,B 90.000,C 0.000} C_DIS
LIN {X 42.762,Y -40.517,Z -141.555,A -90.000,B 90.000,C 0.000} C_DIS
LIN {X 43.078,Y -40.516,Z -141.121,A -90.000,B 90.000,C 0.000} C_DIS
LIN {X 43.227,Y -40.512,Z -140.907,A -90.000,B 90.000,C 0.000} C_DIS
LIN {X 44.071,Y -40.522,Z -139.660,A -90.000,B 90.000,C 0.000} C_DIS
LIN {X 44.134,Y -40.524,Z -139.572,A -90.000,B 90.000,C 0.000} C_DIS
LIN {X 45.156,Y -40.514,Z -138.321,A -90.000,B 90.000,C 0.000} C_DIS
LIN {X 45.282,Y -40.516,Z -138.163,A -90.000,B 90.000,C 0.000} C_DIS
LIN {X 45.824,Y -40.524,Z -137.473,A -90.000,B 90.000,C 0.000} C_DIS
LIN {X 46.601,Y -40.526,Z -136.588,A -90.000,B 90.000,C 0.000} C_DIS
LIN {X 47.252,Y -40.518,Z -135.815,A -90.000,B 90.000,C 0.000} C_DIS
LIN {X 47.463,Y -40.520,Z -135.560,A -90.000,B 90.000,C 0.000} C_DIS
LIN {X 47.738,Y -40.525,Z -135.239,A -90.000,B 90.000,C 0.000} C_DIS
LIN {X 48.146,Y -40.526,Z -134.788,A -90.000,B 90.000,C 0.000} C_DIS
LIN {X 48.676,Y -40.534,Z -134.200,A -90.000,B 90.000,C 0.000} C_DIS
LIN {X 49.622,Y -40.553,Z -133.157,A -90.000,B 90.000,C 0.000} C_DIS
LIN {X 50.350,Y -40.576,Z -132.390,A -90.000,B 90.000,C 0.000} C_DIS
LIN {X 52.547,Y -40.577,Z -129.822,A -90.000,B 90.000,C 0.000} C_DIS
LIN {X 53.228,Y -40.630,Z -128.995,A -90.000,B 90.000,C 0.000} C_DIS
LIN {X 54.741,Y -40.638,Z -126.582,A -90.000,B 90.000,C 0.000} C_DIS
LIN {X 55.173,Y -40.637,Z -125.875,A -90.000,B 90.000,C 0.000} C_DIS
LIN {X 55.300,Y -40.634,Z -125.656,A -90.000,B 90.000,C 0.000} C_DIS
LIN {X 56.108,Y -40.638,Z -124.236,A -90.000,B 90.000,C 0.000} C_DIS
LIN {X 56.908,Y -40.623,Z -122.726,A -90.000,B 90.000,C 0.000} C_DIS
LIN {X 57.351,Y -40.609,Z -121.896,A -90.000,B 90.000,C 0.000} C_DIS
LIN {X 57.424,Y -40.610,Z -121.777,A -90.000,B 90.000,C 0.000} C_DIS
LIN {X 57.466,Y -40.608,Z -121.696,A -90.000,B 90.000,C 0.000} C_DIS
LIN {X 57.634,Y -40.605,Z -121.394,A -90.000,B 90.000,C 0.000} C_DIS
LIN {X 59.656,Y -40.599,Z -117.798,A -90.000,B 90.000,C 0.000} C_DIS
LIN {X 59.815,Y -40.593,Z -117.494,A -90.000,B 90.000,C 0.000} C_DIS
LIN {X 60.155,Y -40.588,Z -116.832,A -90.000,B 90.000,C 0.000} C_DIS
LIN {X 60.381,Y -40.587,Z -116.407,A -90.000,B 90.000,C 0.000} C_DIS
LIN {X 61.359,Y -40.570,Z -114.585,A -90.000,B 90.000,C 0.000} C_DIS
LIN {X 61.746,Y -40.563,Z -113.859,A -90.000,B 90.000,C 0.000} C_DIS
LIN {X 62.273,Y -40.559,Z -112.848,A -90.000,B 90.000,C 0.000} C_DIS
LIN {X 62.387,Y -40.553,Z -112.603,A -90.000,B 90.000,C 0.000} C_DIS
LIN {X 63.292,Y -40.519,Z -110.653,A -90.000,B 90.000,C 0.000} C_DIS
LIN {X 63.346,Y -40.516,Z -110.530,A -90.000,B 90.000,C 0.000} C_DIS
LIN {X 63.470,Y -40.514,Z -110.268,A -90.000,B 90.000,C 0.000} C_DIS
LIN {X 64.451,Y -40.521,Z -108.199,A -90.000,B 90.000,C 0.000} C_DIS
LIN {X 64.698,Y -40.532,Z -107.678,A -90.000,B 90.000,C 0.000} C_DIS
LIN {X 65.204,Y -40.547,Z -106.493,A -90.000,B 90.000,C 0.000} C_DIS
LIN {X 65.229,Y -40.546,Z -106.425,A -90.000,B 90.000,C 0.000} C_DIS
LIN {X 65.794,Y -40.573,Z -104.835,A -90.000,B 90.000,C 0.000} C_DIS
LIN {X 65.810,Y -40.578,Z -104.784,A -90.000,B 90.000,C 0.000} C_DIS
LIN {X 65.833,Y -40.584,Z -104.714,A -90.000,B 90.000,C 0.000} C_DIS
LIN {X 66.029,Y -40.620,Z -103.884,A -90.000,B 90.000,C 0.000} C_DIS
LIN {X 66.218,Y -40.657,Z -103.187,A -90.000,B 90.000,C 0.000} C_DIS
LIN {X 66.226,Y -40.658,Z -103.140,A -90.000,B 90.000,C 0.000} C_DIS
LIN {X 66.329,Y -40.669,Z -102.405,A -90.000,B 90.000,C 0.000} C_DIS
LIN {X 66.346,Y -40.682,Z -102.252,A -90.000,B 90.000,C 0.000} C_DIS
LIN {X 66.320,Y -40.705,Z -101.565,A -90.000,B 90.000,C 0.000} C_DIS
LIN {X 66.235,Y -40.688,Z -101.294,A -90.000,B 90.000,C 0.000} C_DIS
LIN {X 65.811,Y -40.679,Z -100.017,A -90.000,B 90.000,C 0.000} C_DIS
LIN {X 65.787,Y -40.677,Z -99.963,A -90.000,B 90.000,C 0.000} C_DIS
LIN {X 65.730,Y -40.670,Z -99.855,A -90.000,B 90.000,C 0.000} C_DIS
LIN {X 65.385,Y -40.654,Z -99.196,A -90.000,B 90.000,C 0.000} C_DIS
LIN {X 65.117,Y -40.648,Z -98.689,A -90.000,B 90.000,C 0.000} C_DIS
LIN {X 64.741,Y -40.642,Z -97.980,A -90.000,B 90.000,C 0.000} C_DIS
LIN {X 64.338,Y -40.647,Z -97.158,A -90.000,B 90.000,C 0.000} C_DIS
LIN {X 64.024,Y -40.635,Z -96.505,A -90.000,B 90.000,C 0.000} C_DIS
LIN {X 63.992,Y -40.634,Z -96.435,A -90.000,B 90.000,C 0.000} C_DIS
LIN {X 63.797,Y -40.632,Z -95.986,A -90.000,B 90.000,C 0.000} C_DIS
LIN {X 63.688,Y -40.629,Z -95.733,A -90.000,B 90.000,C 0.000} C_DIS
LIN {X 63.622,Y -40.629,Z -95.561,A -90.000,B 90.000,C 0.000} C_DIS
LIN {X 63.535,Y -40.633,Z -95.297,A -90.000,B 90.000,C 0.000} C_DIS
LIN {X 63.521,Y -40.635,Z -95.256,A -90.000,B 90.000,C 0.000} C_DIS
LIN {X 63.496,Y -40.636,Z -95.165,A -90.000,B 90.000,C 0.000} C_DIS
LIN {X 63.458,Y -40.641,Z -95.020,A -90.000,B 90.000,C 0.000} C_DIS
LIN {X 63.363,Y -40.651,Z -94.652,A -90.000,B 90.000,C 0.000} C_DIS
LIN {X 63.078,Y -40.664,Z -93.522,A -90.000,B 90.000,C 0.000} C_DIS
LIN {X 63.010,Y -40.654,Z -93.246,A -90.000,B 90.000,C 0.000} C_DIS
LIN {X 62.833,Y -40.600,Z -92.500,A -90.000,B 90.000,C 0.000} C_DIS
LIN {X 62.793,Y -40.589,Z -92.277,A -90.000,B 90.000,C 0.000} C_DIS
LIN {X 62.758,Y -40.580,Z -91.992,A -90.000,B 90.000,C 0.000} C_DIS
LIN {X 62.735,Y -40.581,Z -91.811,A -90.000,B 90.000,C 0.000} C_DIS
LIN {X 62.724,Y -40.582,Z -91.701,A -90.000,B 90.000,C 0.000} C_DIS
LIN {X 62.718,Y -40.586,Z -91.563,A -90.000,B 90.000,C 0.000} C_DIS
LIN {X 62.718,Y -40.588,Z -91.499,A -90.000,B 90.000,C 0.000} C_DIS
LIN {X 62.719,Y -40.586,Z -91.403,A -90.000,B 90.000,C 0.000} C_DIS
LIN {X 62.719,Y -40.576,Z -91.104,A -90.000,B 90.000,C 0.000} C_DIS
LIN {X 62.701,Y -40.591,Z -89.690,A -90.000,B 90.000,C 0.000} C_DIS
LIN {X 62.700,Y -40.587,Z -89.377,A -90.000,B 90.000,C 0.000} C_DIS
LIN {X 62.706,Y -40.539,Z -88.023,A -90.000,B 90.000,C 0.000} C_DIS
LIN {X 62.709,Y -40.536,Z -87.931,A -90.000,B 90.000,C 0.000} C_DIS
LIN {X 62.717,Y -40.538,Z -87.663,A -90.000,B 90.000,C 0.000} C_DIS
LIN {X 62.744,Y -40.545,Z -87.025,A -90.000,B 90.000,C 0.000} C_DIS
LIN {X 62.779,Y -40.576,Z -86.057,A -90.000,B 90.000,C 0.000} C_DIS
LIN {X 62.777,Y -40.577,Z -85.957,A -90.000,B 90.000,C 0.000} C_DIS
LIN {X 62.745,Y -40.585,Z -84.515,A -90.000,B 90.000,C 0.000} C_DIS
LIN {X 62.754,Y -40.595,Z -84.179,A -90.000,B 90.000,C 0.000} C_DIS
LIN {X 62.764,Y -40.602,Z -84.027,A -90.000,B 90.000,C 0.000} C_DIS
LIN {X 62.775,Y -40.608,Z -83.919,A -90.000,B 90.000,C 0.000} C_DIS
LIN {X 62.775,Y -40.611,Z -83.782,A -90.000,B 90.000,C 0.000} C_DIS
LIN {X 62.768,Y -40.635,Z -83.088,A -90.000,B 90.000,C 0.000} C_DIS
LIN {X 62.755,Y -40.677,Z -82.558,A -90.000,B 90.000,C 0.000} C_DIS
LIN {X 62.732,Y -40.694,Z -82.279,A -90.000,B 90.000,C 0.000} C_DIS
LIN {X 62.670,Y -40.747,Z -81.493,A -90.000,B 90.000,C 0.000} C_DIS
LIN {X 62.637,Y -40.772,Z -81.058,A -90.000,B 90.000,C 0.000} C_DIS
LIN {X 62.492,Y -40.771,Z -80.521,A -90.000,B 90.000,C 0.000} C_DIS
LIN {X 62.469,Y -40.772,Z -80.425,A -90.000,B 90.000,C 0.000} C_DIS
LIN {X 62.458,Y -40.773,Z -80.368,A -90.000,B 90.000,C 0.000} C_DIS
LIN {X 62.437,Y -40.785,Z -80.257,A -90.000,B 90.000,C 0.000} C_DIS
LIN {X 62.390,Y -40.823,Z -79.946,A -90.000,B 90.000,C 0.000} C_DIS
LIN {X 62.315,Y -40.909,Z -79.272,A -90.000,B 90.000,C 0.000} C_DIS
LIN {X 62.296,Y -40.939,Z -79.047,A -90.000,B 90.000,C 0.000} C_DIS
LIN {X 62.292,Y -40.980,Z -78.760,A -90.000,B 90.000,C 0.000} C_DIS
LIN {X 62.303,Y -40.999,Z -78.642,A -90.000,B 90.000,C 0.000} C_DIS
LIN {X 62.349,Y -41.062,Z -78.266,A -90.000,B 90.000,C 0.000} C_DIS
LIN {X 62.372,Y -41.087,Z -78.123,A -90.000,B 90.000,C 0.000} C_DIS
LIN {X 62.395,Y -41.105,Z -78.012,A -90.000,B 90.000,C 0.000} C_DIS
LIN {X 62.101,Y -41.122,Z -77.497,A -90.000,B 90.000,C 0.000} C_DIS
LIN {X 62.034,Y -41.113,Z -77.493,A -90.000,B 90.000,C 0.000} C_DIS
LIN {X 61.582,Y -41.082,Z -77.466,A -90.000,B 90.000,C 0.000} C_DIS
LIN {X 61.492,Y -41.077,Z -77.456,A -90.000,B 90.000,C 0.000} C_DIS
LIN {X 61.083,Y -41.051,Z -77.404,A -90.000,B 90.000,C 0.000} C_DIS
LIN {X 60.787,Y -41.036,Z -77.339,A -90.000,B 90.000,C 0.000} C_DIS
LIN {X 60.643,Y -41.015,Z -77.377,A -90.000,B 90.000,C 0.000} C_DIS
LIN {X 60.470,Y -40.991,Z -77.416,A -90.000,B 90.000,C 0.000} C_DIS
LIN {X 60.171,Y -40.955,Z -77.457,A -90.000,B 90.000,C 0.000} C_DIS
LIN {X 59.518,Y -40.887,Z -77.522,A -90.000,B 90.000,C 0.000} C_DIS
LIN {X 59.281,Y -40.875,Z -77.548,A -90.000,B 90.000,C 0.000} C_DIS
LIN {X 59.140,Y -40.870,Z -77.558,A -90.000,B 90.000,C 0.000} C_DIS
LIN {X 59.028,Y -40.868,Z -77.560,A -90.000,B 90.000,C 0.000} C_DIS
LIN {X 58.342,Y -40.860,Z -77.567,A -90.000,B 90.000,C 0.000} C_DIS
LIN {X 57.312,Y -40.805,Z -77.781,A -90.000,B 90.000,C 0.000} C_DIS
LIN {X 56.914,Y -40.794,Z -77.865,A -90.000,B 90.000,C 0.000} C_DIS
LIN {X 56.672,Y -40.788,Z -77.912,A -90.000,B 90.000,C 0.000} C_DIS
LIN {X 55.855,Y -40.799,Z -78.074,A -90.000,B 90.000,C 0.000} C_DIS
LIN {X 55.106,Y -40.780,Z -78.339,A -90.000,B 90.000,C 0.000} C_DIS
LIN {X 54.825,Y -40.773,Z -78.436,A -90.000,B 90.000,C 0.000} C_DIS
LIN {X 54.700,Y -40.771,Z -78.477,A -90.000,B 90.000,C 0.000} C_DIS
LIN {X 53.933,Y -40.800,Z -78.740,A -90.000,B 90.000,C 0.000} C_DIS
LIN {X 52.253,Y -40.865,Z -79.313,A -90.000,B 90.000,C 0.000} C_DIS
LIN {X 51.497,Y -40.896,Z -79.554,A -90.000,B 90.000,C 0.000} C_DIS
LIN {X 50.871,Y -40.911,Z -79.809,A -90.000,B 90.000,C 0.000} C_DIS
LIN {X 50.581,Y -40.949,Z -79.933,A -90.000,B 90.000,C 0.000} C_DIS
LIN {X 49.566,Y -41.070,Z -80.360,A -90.000,B 90.000,C 0.000} C_DIS
LIN {X 49.497,Y -41.083,Z -80.467,A -90.000,B 90.000,C 0.000} C_DIS
LIN {X 49.660,Y -41.083,Z -80.678,A -90.000,B 90.000,C 0.000} C_DIS
LIN {X 49.736,Y -41.080,Z -80.776,A -90.000,B 90.000,C 0.000} C_DIS
LIN {X 49.788,Y -41.076,Z -80.850,A -90.000,B 90.000,C 0.000} C_DIS
LIN {X 49.846,Y -41.070,Z -80.942,A -90.000,B 90.000,C 0.000} C_DIS
LIN {X 49.909,Y -41.062,Z -81.059,A -90.000,B 90.000,C 0.000} C_DIS
LIN {X 50.013,Y -41.049,Z -81.289,A -90.000,B 90.000,C 0.000} C_DIS
LIN {X 50.083,Y -41.041,Z -81.461,A -90.000,B 90.000,C 0.000} C_DIS
LIN {X 50.114,Y -41.037,Z -81.558,A -90.000,B 90.000,C 0.000} C_DIS
LIN {X 50.175,Y -41.030,Z -81.841,A -90.000,B 90.000,C 0.000} C_DIS
LIN {X 50.201,Y -41.028,Z -82.022,A -90.000,B 90.000,C 0.000} C_DIS
LIN {X 50.213,Y -41.027,Z -82.123,A -90.000,B 90.000,C 0.000} C_DIS
LIN {X 50.224,Y -41.027,Z -82.299,A -90.000,B 90.000,C 0.000} C_DIS
LIN {X 50.358,Y -41.009,Z -82.463,A -90.000,B 90.000,C 0.000} C_DIS
LIN {X 50.463,Y -40.995,Z -82.609,A -90.000,B 90.000,C 0.000} C_DIS
LIN {X 50.476,Y -40.995,Z -82.628,A -90.000,B 90.000,C 0.000} C_DIS
LIN {X 50.574,Y -40.993,Z -82.796,A -90.000,B 90.000,C 0.000} C_DIS
LIN {X 51.367,Y -40.994,Z -84.317,A -90.000,B 90.000,C 0.000} C_DIS
LIN {X 51.410,Y -40.992,Z -84.373,A -90.000,B 90.000,C 0.000} C_DIS
LIN {X 52.241,Y -40.930,Z -85.531,A -90.000,B 90.000,C 0.000} C_DIS
LIN {X 52.421,Y -40.928,Z -85.779,A -90.000,B 90.000,C 0.000} C_DIS
LIN {X 52.489,Y -40.928,Z -85.879,A -90.000,B 90.000,C 0.000} C_DIS
LIN {X 52.658,Y -40.928,Z -86.167,A -90.000,B 90.000,C 0.000} C_DIS
LIN {X 53.306,Y -40.930,Z -87.291,A -90.000,B 90.000,C 0.000} C_DIS
LIN {X 53.445,Y -40.924,Z -87.460,A -90.000,B 90.000,C 0.000} C_DIS
LIN {X 53.584,Y -40.920,Z -87.652,A -90.000,B 90.000,C 0.000} C_DIS
LIN {X 53.668,Y -40.919,Z -87.784,A -90.000,B 90.000,C 0.000} C_DIS
LIN {X 54.570,Y -40.874,Z -89.209,A -90.000,B 90.000,C 0.000} C_DIS
LIN {X 54.750,Y -40.872,Z -89.490,A -90.000,B 90.000,C 0.000} C_DIS
LIN {X 54.844,Y -40.872,Z -89.649,A -90.000,B 90.000,C 0.000} C_DIS
LIN {X 54.909,Y -40.870,Z -89.761,A -90.000,B 90.000,C 0.000} C_DIS
LIN {X 54.973,Y -40.868,Z -89.882,A -90.000,B 90.000,C 0.000} C_DIS
LIN {X 55.796,Y -40.891,Z -91.670,A -90.000,B 90.000,C 0.000} C_DIS
LIN {X 55.881,Y -40.886,Z -91.859,A -90.000,B 90.000,C 0.000} C_DIS
LIN {X 55.925,Y -40.883,Z -91.946,A -90.000,B 90.000,C 0.000} C_DIS
LIN {X 56.026,Y -40.878,Z -92.200,A -90.000,B 90.000,C 0.000} C_DIS
LIN {X 56.124,Y -40.877,Z -92.503,A -90.000,B 90.000,C 0.000} C_DIS
LIN {X 56.440,Y -40.880,Z -93.570,A -90.000,B 90.000,C 0.000} C_DIS
LIN {X 56.501,Y -40.882,Z -93.777,A -90.000,B 90.000,C 0.000} C_DIS
LIN {X 56.580,Y -40.884,Z -94.042,A -90.000,B 90.000,C 0.000} C_DIS
LIN {X 56.765,Y -40.862,Z -94.689,A -90.000,B 90.000,C 0.000} C_DIS
LIN {X 57.395,Y -40.787,Z -96.896,A -90.000,B 90.000,C 0.000} C_DIS
LIN {X 57.428,Y -40.784,Z -97.061,A -90.000,B 90.000,C 0.000} C_DIS
LIN {X 57.465,Y -40.783,Z -97.319,A -90.000,B 90.000,C 0.000} C_DIS
LIN {X 57.495,Y -40.783,Z -97.620,A -90.000,B 90.000,C 0.000} C_DIS
LIN {X 57.500,Y -40.785,Z -97.716,A -90.000,B 90.000,C 0.000} C_DIS
LIN {X 57.583,Y -40.788,Z -98.631,A -90.000,B 90.000,C 0.000} C_DIS
LIN {X 57.585,Y -40.787,Z -98.670,A -90.000,B 90.000,C 0.000} C_DIS
LIN {X 57.670,Y -40.741,Z -100.908,A -90.000,B 90.000,C 0.000} C_DIS
LIN {X 57.687,Y -40.721,Z -101.434,A -90.000,B 90.000,C 0.000} C_DIS
LIN {X 57.686,Y -40.716,Z -101.554,A -90.000,B 90.000,C 0.000} C_DIS
LIN {X 57.680,Y -40.710,Z -101.694,A -90.000,B 90.000,C 0.000} C_DIS
LIN {X 57.669,Y -40.703,Z -101.841,A -90.000,B 90.000,C 0.000} C_DIS
LIN {X 57.592,Y -40.677,Z -102.538,A -90.000,B 90.000,C 0.000} C_DIS
LIN {X 57.446,Y -40.667,Z -103.992,A -90.000,B 90.000,C 0.000} C_DIS
LIN {X 57.418,Y -40.661,Z -104.251,A -90.000,B 90.000,C 0.000} C_DIS
LIN {X 57.403,Y -40.654,Z -104.381,A -90.000,B 90.000,C 0.000} C_DIS
LIN {X 57.328,Y -40.573,Z -105.504,A -90.000,B 90.000,C 0.000} C_DIS
LIN {X 57.301,Y -40.562,Z -105.728,A -90.000,B 90.000,C 0.000} C_DIS
LIN {X 57.218,Y -40.549,Z -106.204,A -90.000,B 90.000,C 0.000} C_DIS
LIN {X 57.043,Y -40.541,Z -107.256,A -90.000,B 90.000,C 0.000} C_DIS
LIN {X 57.015,Y -40.535,Z -107.411,A -90.000,B 90.000,C 0.000} C_DIS
LIN {X 56.586,Y -40.457,Z -109.629,A -90.000,B 90.000,C 0.000} C_DIS
LIN {X 56.552,Y -40.454,Z -109.778,A -90.000,B 90.000,C 0.000} C_DIS
LIN {X 56.442,Y -40.449,Z -110.221,A -90.000,B 90.000,C 0.000} C_DIS
LIN {X 55.898,Y -40.411,Z -112.375,A -90.000,B 90.000,C 0.000} C_DIS
LIN {X 55.805,Y -40.408,Z -112.719,A -90.000,B 90.000,C 0.000} C_DIS
LIN {X 55.444,Y -40.386,Z -113.882,A -90.000,B 90.000,C 0.000} C_DIS
LIN {X 54.963,Y -40.365,Z -115.303,A -90.000,B 90.000,C 0.000} C_DIS
LIN {X 54.886,Y -40.361,Z -115.527,A -90.000,B 90.000,C 0.000} C_DIS
LIN {X 54.651,Y -40.357,Z -116.155,A -90.000,B 90.000,C 0.000} C_DIS
LIN {X 54.060,Y -40.330,Z -117.700,A -90.000,B 90.000,C 0.000} C_DIS
LIN {X 53.993,Y -40.329,Z -117.865,A -90.000,B 90.000,C 0.000} C_DIS
LIN {X 53.906,Y -40.330,Z -118.070,A -90.000,B 90.000,C 0.000} C_DIS
LIN {X 53.532,Y -40.318,Z -118.883,A -90.000,B 90.000,C 0.000} C_DIS
LIN {X 53.326,Y -40.304,Z -119.321,A -90.000,B 90.000,C 0.000} C_DIS
LIN {X 52.608,Y -40.278,Z -120.765,A -90.000,B 90.000,C 0.000} C_DIS
LIN {X 52.281,Y -40.271,Z -121.428,A -90.000,B 90.000,C 0.000} C_DIS
LIN {X 52.115,Y -40.261,Z -121.752,A -90.000,B 90.000,C 0.000} C_DIS
LIN {X 51.964,Y -40.261,Z -122.016,A -90.000,B 90.000,C 0.000} C_DIS
LIN {X 51.910,Y -40.259,Z -122.108,A -90.000,B 90.000,C 0.000} C_DIS
LIN {X 51.625,Y -40.246,Z -122.555,A -90.000,B 90.000,C 0.000} C_DIS
LIN {X 50.470,Y -40.222,Z -124.288,A -90.000,B 90.000,C 0.000} C_DIS
LIN {X 49.747,Y -40.193,Z -125.350,A -90.000,B 90.000,C 0.000} C_DIS
LIN {X 49.625,Y -40.190,Z -125.523,A -90.000,B 90.000,C 0.000} C_DIS
LIN {X 49.517,Y -40.186,Z -125.668,A -90.000,B 90.000,C 0.000} C_DIS
LIN {X 49.397,Y -40.185,Z -125.820,A -90.000,B 90.000,C 0.000} C_DIS
LIN {X 49.333,Y -40.181,Z -125.897,A -90.000,B 90.000,C 0.000} C_DIS
LIN {X 49.216,Y -40.175,Z -126.032,A -90.000,B 90.000,C 0.000} C_DIS
LIN {X 46.887,Y -40.138,Z -128.545,A -90.000,B 90.000,C 0.000} C_DIS
LIN {X 46.604,Y -40.130,Z -128.846,A -90.000,B 90.000,C 0.000} C_DIS
LIN {X 46.441,Y -40.122,Z -129.017,A -90.000,B 90.000,C 0.000} C_DIS
LIN {X 46.357,Y -40.120,Z -129.100,A -90.000,B 90.000,C 0.000} C_DIS
LIN {X 46.097,Y -40.110,Z -129.337,A -90.000,B 90.000,C 0.000} C_DIS
LIN {X 45.337,Y -40.088,Z -130.013,A -90.000,B 90.000,C 0.000} C_DIS
LIN {X 43.243,Y -40.061,Z -131.818,A -90.000,B 90.000,C 0.000} C_DIS
LIN {X 42.942,Y -40.047,Z -132.067,A -90.000,B 90.000,C 0.000} C_DIS
LIN {X 41.761,Y -40.027,Z -132.995,A -90.000,B 90.000,C 0.000} C_DIS
LIN {X 39.773,Y -40.007,Z -134.481,A -90.000,B 90.000,C 0.000} C_DIS
LIN {X 37.609,Y -39.967,Z -136.061,A -90.000,B 90.000,C 0.000} C_DIS
LIN {X 36.596,Y -39.938,Z -136.784,A -90.000,B 90.000,C 0.000} C_DIS
LIN {X 36.286,Y -39.938,Z -137.003,A -90.000,B 90.000,C 0.000} C_DIS
LIN {X 34.393,Y -39.899,Z -138.379,A -90.000,B 90.000,C 0.000} C_DIS
LIN {X 33.503,Y -39.883,Z -139.020,A -90.000,B 90.000,C 0.000} C_DIS
LIN {X 33.227,Y -39.879,Z -139.222,A -90.000,B 90.000,C 0.000} C_DIS
LIN {X 32.658,Y -39.881,Z -139.623,A -90.000,B 90.000,C 0.000} C_DIS
LIN {X 30.670,Y -39.858,Z -140.985,A -90.000,B 90.000,C 0.000} C_DIS
LIN {X 30.325,Y -39.846,Z -141.231,A -90.000,B 90.000,C 0.000} C_DIS
LIN {X 30.206,Y -39.840,Z -141.313,A -90.000,B 90.000,C 0.000} C_DIS
LIN {X 30.104,Y -39.838,Z -141.380,A -90.000,B 90.000,C 0.000} C_DIS
LIN {X 29.038,Y -39.842,Z -142.056,A -90.000,B 90.000,C 0.000} C_DIS
LIN {X 27.597,Y -39.834,Z -142.951,A -90.000,B 90.000,C 0.000} C_DIS
LIN {X 26.950,Y -39.819,Z -143.362,A -90.000,B 90.000,C 0.000} C_DIS
LIN {X 26.698,Y -39.815,Z -143.518,A -90.000,B 90.000,C 0.000} C_DIS
LIN {X 26.480,Y -39.805,Z -143.642,A -90.000,B 90.000,C 0.000} C_DIS
LIN {X 26.392,Y -39.804,Z -143.690,A -90.000,B 90.000,C 0.000} C_DIS
LIN {X 24.352,Y -39.811,Z -144.770,A -90.000,B 90.000,C 0.000} C_DIS
LIN {X 22.834,Y -39.820,Z -145.576,A -90.000,B 90.000,C 0.000} C_DIS
LIN {X 22.635,Y -39.819,Z -145.678,A -90.000,B 90.000,C 0.000} C_DIS
LIN {X 22.456,Y -39.816,Z -145.767,A -90.000,B 90.000,C 0.000} C_DIS
LIN {X 22.256,Y -39.817,Z -145.863,A -90.000,B 90.000,C 0.000} C_DIS
LIN {X 22.039,Y -39.816,Z -145.962,A -90.000,B 90.000,C 0.000} C_DIS
LIN {X 21.929,Y -39.818,Z -146.010,A -90.000,B 90.000,C 0.000} C_DIS
LIN {X 21.754,Y -39.825,Z -146.082,A -90.000,B 90.000,C 0.000} C_DIS
LIN {X 21.166,Y -39.840,Z -146.311,A -90.000,B 90.000,C 0.000} C_DIS
LIN {X 19.940,Y -39.863,Z -146.779,A -90.000,B 90.000,C 0.000} C_DIS
LIN {X 19.289,Y -39.859,Z -147.008,A -90.000,B 90.000,C 0.000} C_DIS
LIN {X 18.452,Y -39.857,Z -147.298,A -90.000,B 90.000,C 0.000} C_DIS
LIN {X 17.955,Y -39.854,Z -147.469,A -90.000,B 90.000,C 0.000} C_DIS
LIN {X 17.327,Y -39.848,Z -147.682,A -90.000,B 90.000,C 0.000} C_DIS
LIN {X 16.996,Y -39.850,Z -147.790,A -90.000,B 90.000,C 0.000} C_DIS
LIN {X 16.265,Y -39.850,Z -148.020,A -90.000,B 90.000,C 0.000} C_DIS
LIN {X 15.173,Y -39.884,Z -148.330,A -90.000,B 90.000,C 0.000} C_DIS
LIN {X 14.231,Y -39.910,Z -148.592,A -90.000,B 90.000,C 0.000} C_DIS
LIN {X 13.439,Y -39.914,Z -148.794,A -90.000,B 90.000,C 0.000} C_DIS
LIN {X 12.800,Y -39.911,Z -148.951,A -90.000,B 90.000,C 0.000} C_DIS
LIN {X 11.387,Y -39.894,Z -149.286,A -90.000,B 90.000,C 0.000} C_DIS
LIN {X 10.876,Y -39.902,Z -149.392,A -90.000,B 90.000,C 0.000} C_DIS
LIN {X 9.877,Y -39.938,Z -149.579,A -90.000,B 90.000,C 0.000} C_DIS
LIN {X 9.402,Y -39.950,Z -149.659,A -90.000,B 90.000,C 0.000} C_DIS
LIN {X 8.997,Y -39.951,Z -149.719,A -90.000,B 90.000,C 0.000} C_DIS
LIN {X 7.388,Y -39.933,Z -149.936,A -90.000,B 90.000,C 0.000} C_DIS
LIN {X 7.054,Y -39.931,Z -149.979,A -90.000,B 90.000,C 0.000} C_DIS
LIN {X 6.442,Y -39.922,Z -150.051,A -90.000,B 90.000,C 0.000} C_DIS
LIN {X 5.965,Y -39.931,Z -150.092,A -90.000,B 90.000,C 0.000} C_DIS
LIN {X 5.265,Y -39.959,Z -150.138,A -90.000,B 90.000,C 0.000} C_DIS
LIN {X 4.869,Y -39.966,Z -150.155,A -90.000,B 90.000,C 0.000} C_DIS
LIN {X 3.721,Y -39.957,Z -150.177,A -90.000,B 90.000,C 0.000} C_DIS
LIN {X 1.825,Y -39.930,Z -150.185,A -90.000,B 90.000,C 0.000} C_DIS
LIN {X 1.731,Y -39.930,Z -150.184,A -90.000,B 90.000,C 0.000} C_DIS
LIN {X 1.284,Y -39.939,Z -150.171,A -90.000,B 90.000,C 0.000} C_DIS
LIN {X 1.197,Y -39.942,Z -150.167,A -90.000,B 90.000,C 0.000} C_DIS
LIN {X 0.800,Y -39.954,Z -150.131,A -90.000,B 90.000,C 0.000} C_DIS
LIN {X 0.222,Y -39.952,Z -150.056,A -90.000,B 90.000,C 0.000} C_DIS
LIN {X -2.689,Y -39.924,Z -149.649,A -90.000,B 90.000,C 0.000} C_DIS
LIN {X -2.815,Y -39.925,Z -149.629,A -90.000,B 90.000,C 0.000} C_DIS
LIN {X -3.060,Y -39.923,Z -149.586,A -90.000,B 90.000,C 0.000} C_DIS
LIN {X -3.211,Y -39.925,Z -149.555,A -90.000,B 90.000,C 0.000} C_DIS
LIN {X -4.062,Y -39.924,Z -149.317,A -90.000,B 90.000,C 0.000} C_DIS
LIN {X -6.966,Y -39.916,Z -148.499,A -90.000,B 90.000,C 0.000} C_DIS
LIN {X -7.197,Y -39.917,Z -148.430,A -90.000,B 90.000,C 0.000} C_DIS
LIN {X -7.300,Y -39.912,Z -148.393,A -90.000,B 90.000,C 0.000} C_DIS
LIN {X -7.442,Y -39.908,Z -148.338,A -90.000,B 90.000,C 0.000} C_DIS
LIN {X -9.169,Y -39.920,Z -147.610,A -90.000,B 90.000,C 0.000} C_DIS
LIN {X -11.038,Y -39.930,Z -146.816,A -90.000,B 90.000,C 0.000} C_DIS
LIN {X -11.202,Y -39.931,Z -146.744,A -90.000,B 90.000,C 0.000} C_DIS
LIN {X -11.491,Y -39.918,Z -146.597,A -90.000,B 90.000,C 0.000} C_DIS
LIN {X -11.621,Y -39.917,Z -146.527,A -90.000,B 90.000,C 0.000} C_DIS
LIN {X -14.581,Y -39.970,Z -144.831,A -90.000,B 90.000,C 0.000} C_DIS
LIN {X -15.102,Y -39.976,Z -144.525,A -90.000,B 90.000,C 0.000} C_DIS
LIN {X -15.225,Y -39.970,Z -144.442,A -90.000,B 90.000,C 0.000} C_DIS
LIN {X -15.516,Y -39.961,Z -144.242,A -90.000,B 90.000,C 0.000} C_DIS
LIN {X -17.104,Y -39.998,Z -143.050,A -90.000,B 90.000,C 0.000} C_DIS
LIN {X -17.898,Y -40.021,Z -142.415,A -90.000,B 90.000,C 0.000} C_DIS
LIN {X -18.395,Y -40.035,Z -142.013,A -90.000,B 90.000,C 0.000} C_DIS
LIN {X -18.707,Y -40.038,Z -141.756,A -90.000,B 90.000,C 0.000} C_DIS
LIN {X -18.810,Y -40.034,Z -141.665,A -90.000,B 90.000,C 0.000} C_DIS
LIN {X -18.932,Y -40.034,Z -141.551,A -90.000,B 90.000,C 0.000} C_DIS
LIN {X -19.248,Y -40.046,Z -141.238,A -90.000,B 90.000,C 0.000} C_DIS
LIN {X -19.947,Y -40.089,Z -140.519,A -90.000,B 90.000,C 0.000} C_DIS
LIN {X -20.911,Y -40.142,Z -139.516,A -90.000,B 90.000,C 0.000} C_DIS
LIN {X -21.504,Y -40.193,Z -138.867,A -90.000,B 90.000,C 0.000} C_DIS
LIN {X -21.725,Y -40.206,Z -138.616,A -90.000,B 90.000,C 0.000} C_DIS
LIN {X -21.855,Y -40.208,Z -138.463,A -90.000,B 90.000,C 0.000} C_DIS
LIN {X -21.931,Y -40.211,Z -138.369,A -90.000,B 90.000,C 0.000} C_DIS
LIN {X -22.558,Y -40.257,Z -137.551,A -90.000,B 90.000,C 0.000} C_DIS
LIN {X -22.671,Y -40.260,Z -137.397,A -90.000,B 90.000,C 0.000} C_DIS
LIN {X -23.341,Y -40.295,Z -136.447,A -90.000,B 90.000,C 0.000} C_DIS
LIN {X -23.394,Y -40.297,Z -136.369,A -90.000,B 90.000,C 0.000} C_DIS
LIN {X -23.868,Y -40.318,Z -135.654,A -90.000,B 90.000,C 0.000} C_DIS
LIN {X -24.033,Y -40.321,Z -135.401,A -90.000,B 90.000,C 0.000} C_DIS
LIN {X -24.115,Y -40.324,Z -135.268,A -90.000,B 90.000,C 0.000} C_DIS
LIN {X -24.209,Y -40.324,Z -135.109,A -90.000,B 90.000,C 0.000} C_DIS
LIN {X -24.291,Y -40.326,Z -134.965,A -90.000,B 90.000,C 0.000} C_DIS
LIN {X -24.399,Y -40.333,Z -134.757,A -90.000,B 90.000,C 0.000} C_DIS
LIN {X -24.443,Y -40.337,Z -134.668,A -90.000,B 90.000,C 0.000} C_DIS
LIN {X -24.834,Y -40.389,Z -133.828,A -90.000,B 90.000,C 0.000} C_DIS
LIN {X -25.464,Y -40.499,Z -132.361,A -90.000,B 90.000,C 0.000} C_DIS
LIN {X -25.499,Y -40.507,Z -132.275,A -90.000,B 90.000,C 0.000} C_DIS
LIN {X -25.732,Y -40.549,Z -131.685,A -90.000,B 90.000,C 0.000} C_DIS
LIN {X -25.950,Y -40.581,Z -131.119,A -90.000,B 90.000,C 0.000} C_DIS
LIN {X -26.202,Y -40.591,Z -130.433,A -90.000,B 90.000,C 0.000} C_DIS
LIN {X -26.427,Y -40.587,Z -129.902,A -90.000,B 90.000,C 0.000} C_DIS
LIN {X -26.753,Y -40.571,Z -129.122,A -90.000,B 90.000,C 0.000} C_DIS
LIN {X -26.804,Y -40.571,Z -128.989,A -90.000,B 90.000,C 0.000} C_DIS
LIN {X -26.902,Y -40.580,Z -128.698,A -90.000,B 90.000,C 0.000} C_DIS
LIN {X -26.979,Y -40.592,Z -128.446,A -90.000,B 90.000,C 0.000} C_DIS
LIN {X -27.153,Y -40.607,Z -127.839,A -90.000,B 90.000,C 0.000} C_DIS
LIN {X -27.178,Y -40.610,Z -127.745,A -90.000,B 90.000,C 0.000} C_DIS
LIN {X -27.252,Y -40.614,Z -127.510,A -90.000,B 90.000,C 0.000} C_DIS
LIN {X -27.317,Y -40.618,Z -127.291,A -90.000,B 90.000,C 0.000} C_DIS
LIN {X -27.645,Y -40.682,Z -126.234,A -90.000,B 90.000,C 0.000} C_DIS
LIN {X -28.117,Y -40.689,Z -125.118,A -90.000,B 90.000,C 0.000} C_DIS
LIN {X -28.266,Y -40.679,Z -124.755,A -90.000,B 90.000,C 0.000} C_DIS
LIN {X -28.432,Y -40.664,Z -124.348,A -90.000,B 90.000,C 0.000} C_DIS
LIN {X -28.487,Y -40.661,Z -124.197,A -90.000,B 90.000,C 0.000} C_DIS
LIN {X -28.834,Y -40.652,Z -123.109,A -90.000,B 90.000,C 0.000} C_DIS
LIN {X -29.170,Y -40.714,Z -121.950,A -90.000,B 90.000,C 0.000} C_DIS
LIN {X -29.300,Y -40.714,Z -121.657,A -90.000,B 90.000,C 0.000} C_DIS
LIN {X -29.393,Y -40.706,Z -121.442,A -90.000,B 90.000,C 0.000} C_DIS
LIN {X -29.772,Y -40.673,Z -120.563,A -90.000,B 90.000,C 0.000} C_DIS
LIN {X -29.841,Y -40.663,Z -120.400,A -90.000,B 90.000,C 0.000} C_DIS
LIN {X -29.898,Y -40.656,Z -120.248,A -90.000,B 90.000,C 0.000} C_DIS
LIN {X -30.026,Y -40.645,Z -119.845,A -90.000,B 90.000,C 0.000} C_DIS
LIN {X -30.058,Y -40.644,Z -119.736,A -90.000,B 90.000,C 0.000} C_DIS
LIN {X -30.160,Y -40.641,Z -119.343,A -90.000,B 90.000,C 0.000} C_DIS
LIN {X -30.204,Y -40.649,Z -119.183,A -90.000,B 90.000,C 0.000} C_DIS
LIN {X -30.507,Y -40.710,Z -118.044,A -90.000,B 90.000,C 0.000} C_DIS
LIN {X -30.678,Y -40.710,Z -117.637,A -90.000,B 90.000,C 0.000} C_DIS
LIN {X -30.812,Y -40.700,Z -117.310,A -90.000,B 90.000,C 0.000} C_DIS
LIN {X -31.026,Y -40.654,Z -116.760,A -90.000,B 90.000,C 0.000} C_DIS
LIN {X -31.044,Y -40.650,Z -116.714,A -90.000,B 90.000,C 0.000} C_DIS
LIN {X -31.250,Y -40.603,Z -116.134,A -90.000,B 90.000,C 0.000} C_DIS
LIN {X -31.346,Y -40.583,Z -115.836,A -90.000,B 90.000,C 0.000} C_DIS
LIN {X -31.390,Y -40.575,Z -115.679,A -90.000,B 90.000,C 0.000} C_DIS
LIN {X -31.416,Y -40.572,Z -115.568,A -90.000,B 90.000,C 0.000} C_DIS
LIN {X -31.514,Y -40.579,Z -115.188,A -90.000,B 90.000,C 0.000} C_DIS
LIN {X -31.555,Y -40.587,Z -114.992,A -90.000,B 90.000,C 0.000} C_DIS
LIN {X -31.617,Y -40.610,Z -114.594,A -90.000,B 90.000,C 0.000} C_DIS
LIN {X -31.711,Y -40.641,Z -113.972,A -90.000,B 90.000,C 0.000} C_DIS
LIN {X -31.743,Y -40.642,Z -113.726,A -90.000,B 90.000,C 0.000} C_DIS
LIN {X -31.768,Y -40.638,Z -113.614,A -90.000,B 90.000,C 0.000} C_DIS
LIN {X -31.911,Y -40.638,Z -112.994,A -90.000,B 90.000,C 0.000} C_DIS
LIN {X -31.930,Y -40.637,Z -112.878,A -90.000,B 90.000,C 0.000} C_DIS
LIN {X -31.969,Y -40.638,Z -112.598,A -90.000,B 90.000,C 0.000} C_DIS
LIN {X -31.979,Y -40.639,Z -112.516,A -90.000,B 90.000,C 0.000} C_DIS
LIN {X -32.035,Y -40.650,Z -111.950,A -90.000,B 90.000,C 0.000} C_DIS
LIN {X -32.072,Y -40.644,Z -111.541,A -90.000,B 90.000,C 0.000} C_DIS
LIN {X -32.083,Y -40.643,Z -111.463,A -90.000,B 90.000,C 0.000} C_DIS
LIN {X -32.141,Y -40.630,Z -111.067,A -90.000,B 90.000,C 0.000} C_DIS
LIN {X -32.279,Y -40.563,Z -110.024,A -90.000,B 90.000,C 0.000} C_DIS
LIN {X -32.317,Y -40.544,Z -109.690,A -90.000,B 90.000,C 0.000} C_DIS
LIN {X -32.329,Y -40.538,Z -109.555,A -90.000,B 90.000,C 0.000} C_DIS
LIN {X -32.357,Y -40.532,Z -109.163,A -90.000,B 90.000,C 0.000} C_DIS
LIN {X -32.359,Y -40.533,Z -109.050,A -90.000,B 90.000,C 0.000} C_DIS
LIN {X -32.350,Y -40.543,Z -108.718,A -90.000,B 90.000,C 0.000} C_DIS
LIN {X -32.330,Y -40.559,Z -108.286,A -90.000,B 90.000,C 0.000} C_DIS
LIN {X -32.267,Y -40.567,Z -107.239,A -90.000,B 90.000,C 0.000} C_DIS
LIN {X -32.259,Y -40.567,Z -107.007,A -90.000,B 90.000,C 0.000} C_DIS
LIN {X -32.244,Y -40.566,Z -106.571,A -90.000,B 90.000,C 0.000} C_DIS
LIN {X -32.234,Y -40.563,Z -106.419,A -90.000,B 90.000,C 0.000} C_DIS
LIN {X -32.221,Y -40.563,Z -106.267,A -90.000,B 90.000,C 0.000} C_DIS
LIN {X -32.156,Y -40.549,Z -105.601,A -90.000,B 90.000,C 0.000} C_DIS
LIN {X -32.122,Y -40.535,Z -105.290,A -90.000,B 90.000,C 0.000} C_DIS
LIN {X -32.044,Y -40.489,Z -104.411,A -90.000,B 90.000,C 0.000} C_DIS
LIN {X -32.002,Y -40.465,Z -103.929,A -90.000,B 90.000,C 0.000} C_DIS
LIN {X -31.968,Y -40.453,Z -103.589,A -90.000,B 90.000,C 0.000} C_DIS
LIN {X -31.906,Y -40.418,Z -102.823,A -90.000,B 90.000,C 0.000} C_DIS
LIN {X -31.867,Y -40.407,Z -102.490,A -90.000,B 90.000,C 0.000} C_DIS
LIN {X -31.813,Y -40.397,Z -102.021,A -90.000,B 90.000,C 0.000} C_DIS
LIN {X -31.749,Y -40.383,Z -101.477,A -90.000,B 90.000,C 0.000} C_DIS
LIN {X -31.732,Y -40.382,Z -101.356,A -90.000,B 90.000,C 0.000} C_DIS
LIN {X -31.597,Y -40.391,Z -100.661,A -90.000,B 90.000,C 0.000} C_DIS
LIN {X -31.573,Y -40.391,Z -100.540,A -90.000,B 90.000,C 0.000} C_DIS
LIN {X -31.489,Y -40.387,Z -100.136,A -90.000,B 90.000,C 0.000} C_DIS
LIN {X -31.373,Y -40.372,Z -99.601,A -90.000,B 90.000,C 0.000} C_DIS
LIN {X -31.237,Y -40.345,Z -98.913,A -90.000,B 90.000,C 0.000} C_DIS
LIN {X -31.209,Y -40.342,Z -98.790,A -90.000,B 90.000,C 0.000} C_DIS
LIN {X -31.120,Y -40.339,Z -98.443,A -90.000,B 90.000,C 0.000} C_DIS
LIN {X -30.996,Y -40.339,Z -97.953,A -90.000,B 90.000,C 0.000} C_DIS
LIN {X -30.966,Y -40.336,Z -97.839,A -90.000,B 90.000,C 0.000} C_DIS
LIN {X -30.799,Y -40.311,Z -97.162,A -90.000,B 90.000,C 0.000} C_DIS
LIN {X -30.634,Y -40.296,Z -96.468,A -90.000,B 90.000,C 0.000} C_DIS
LIN {X -30.543,Y -40.292,Z -96.114,A -90.000,B 90.000,C 0.000} C_DIS
LIN {X -30.504,Y -40.294,Z -95.980,A -90.000,B 90.000,C 0.000} C_DIS
LIN {X -30.390,Y -40.304,Z -95.622,A -90.000,B 90.000,C 0.000} C_DIS
LIN {X -30.075,Y -40.283,Z -94.651,A -90.000,B 90.000,C 0.000} C_DIS
LIN {X -29.776,Y -40.279,Z -93.799,A -90.000,B 90.000,C 0.000} C_DIS
LIN {X -29.714,Y -40.281,Z -93.630,A -90.000,B 90.000,C 0.000} C_DIS
LIN {X -29.594,Y -40.289,Z -93.337,A -90.000,B 90.000,C 0.000} C_DIS
LIN {X -29.038,Y -40.316,Z -92.131,A -90.000,B 90.000,C 0.000} C_DIS
LIN {X -28.592,Y -40.326,Z -91.182,A -90.000,B 90.000,C 0.000} C_DIS
LIN {X -28.551,Y -40.328,Z -91.098,A -90.000,B 90.000,C 0.000} C_DIS
LIN {X -27.966,Y -40.367,Z -90.073,A -90.000,B 90.000,C 0.000} C_DIS
LIN {X -27.616,Y -40.377,Z -89.477,A -90.000,B 90.000,C 0.000} C_DIS
LIN {X -27.426,Y -40.377,Z -89.134,A -90.000,B 90.000,C 0.000} C_DIS
LIN {X -27.339,Y -40.378,Z -88.981,A -90.000,B 90.000,C 0.000} C_DIS
LIN {X -27.247,Y -40.382,Z -88.831,A -90.000,B 90.000,C 0.000} C_DIS
LIN {X -27.134,Y -40.384,Z -88.650,A -90.000,B 90.000,C 0.000} C_DIS
LIN {X -26.752,Y -40.407,Z -88.094,A -90.000,B 90.000,C 0.000} C_DIS
LIN {X -26.229,Y -40.427,Z -87.340,A -90.000,B 90.000,C 0.000} C_DIS
LIN {X -25.876,Y -40.436,Z -86.837,A -90.000,B 90.000,C 0.000} C_DIS
LIN {X -25.671,Y -40.440,Z -86.558,A -90.000,B 90.000,C 0.000} C_DIS
LIN {X -25.595,Y -40.443,Z -86.461,A -90.000,B 90.000,C 0.000} C_DIS
LIN {X -25.199,Y -40.468,Z -85.982,A -90.000,B 90.000,C 0.000} C_DIS
LIN {X -24.398,Y -40.498,Z -85.029,A -90.000,B 90.000,C 0.000} C_DIS
LIN {X -24.136,Y -40.511,Z -84.729,A -90.000,B 90.000,C 0.000} C_DIS
LIN {X -23.817,Y -40.516,Z -84.373,A -90.000,B 90.000,C 0.000} C_DIS
LIN {X -23.607,Y -40.520,Z -84.143,A -90.000,B 90.000,C 0.000} C_DIS
LIN {X -22.748,Y -40.551,Z -83.255,A -90.000,B 90.000,C 0.000} C_DIS
LIN {X -22.387,Y -40.557,Z -82.886,A -90.000,B 90.000,C 0.000} C_DIS
LIN {X -22.327,Y -40.559,Z -82.827,A -90.000,B 90.000,C 0.000} C_DIS
LIN {X -21.787,Y -40.581,Z -82.317,A -90.000,B 90.000,C 0.000} C_DIS
LIN {X -21.510,Y -40.586,Z -82.059,A -90.000,B 90.000,C 0.000} C_DIS
LIN {X -21.336,Y -40.585,Z -81.899,A -90.000,B 90.000,C 0.000} C_DIS
LIN {X -21.238,Y -40.586,Z -81.810,A -90.000,B 90.000,C 0.000} C_DIS
LIN {X -20.836,Y -40.594,Z -81.472,A -90.000,B 90.000,C 0.000} C_DIS
LIN {X -20.762,Y -40.596,Z -81.411,A -90.000,B 90.000,C 0.000} C_DIS
LIN {X -20.368,Y -40.613,Z -81.110,A -90.000,B 90.000,C 0.000} C_DIS
LIN {X -19.989,Y -40.623,Z -80.826,A -90.000,B 90.000,C 0.000} C_DIS
LIN {X -19.808,Y -40.630,Z -80.700,A -90.000,B 90.000,C 0.000} C_DIS
LIN {X -19.019,Y -40.646,Z -80.169,A -90.000,B 90.000,C 0.000} C_DIS
LIN {X -18.850,Y -40.643,Z -80.057,A -90.000,B 90.000,C 0.000} C_DIS
LIN {X -18.727,Y -40.643,Z -79.982,A -90.000,B 90.000,C 0.000} C_DIS
LIN {X -18.116,Y -40.653,Z -79.636,A -90.000,B 90.000,C 0.000} C_DIS
LIN {X -17.862,Y -40.650,Z -79.495,A -90.000,B 90.000,C 0.000} C_DIS
LIN {X -17.530,Y -40.651,Z -79.325,A -90.000,B 90.000,C 0.000} C_DIS
LIN {X -16.966,Y -40.661,Z -79.066,A -90.000,B 90.000,C 0.000} C_DIS
LIN {X -16.580,Y -40.661,Z -78.893,A -90.000,B 90.000,C 0.000} C_DIS
LIN {X -16.440,Y -40.662,Z -78.836,A -90.000,B 90.000,C 0.000} C_DIS
LIN {X -16.211,Y -40.669,Z -78.754,A -90.000,B 90.000,C 0.000} C_DIS
LIN {X -15.527,Y -40.669,Z -78.514,A -90.000,B 90.000,C 0.000} C_DIS
LIN {X -15.357,Y -40.671,Z -78.461,A -90.000,B 90.000,C 0.000} C_DIS
LIN {X -15.047,Y -40.671,Z -78.369,A -90.000,B 90.000,C 0.000} C_DIS
LIN {X -14.861,Y -40.667,Z -78.315,A -90.000,B 90.000,C 0.000} C_DIS
LIN {X -14.108,Y -40.649,Z -78.097,A -90.000,B 90.000,C 0.000} C_DIS
LIN {X -13.918,Y -40.643,Z -78.051,A -90.000,B 90.000,C 0.000} C_DIS
LIN {X -13.277,Y -40.633,Z -77.927,A -90.000,B 90.000,C 0.000} C_DIS
LIN {X -12.656,Y -40.614,Z -77.810,A -90.000,B 90.000,C 0.000} C_DIS
LIN {X -12.519,Y -40.611,Z -77.789,A -90.000,B 90.000,C 0.000} C_DIS
LIN {X -12.219,Y -40.610,Z -77.755,A -90.000,B 90.000,C 0.000} C_DIS
LIN {X -11.730,Y -40.610,Z -77.705,A -90.000,B 90.000,C 0.000} C_DIS
LIN {X -11.244,Y -40.600,Z -77.660,A -90.000,B 90.000,C 0.000} C_DIS
LIN {X -11.128,Y -40.599,Z -77.652,A -90.000,B 90.000,C 0.000} C_DIS
LIN {X -10.439,Y -40.599,Z -77.626,A -90.000,B 90.000,C 0.000} C_DIS
LIN {X -10.359,Y -40.599,Z -77.624,A -90.000,B 90.000,C 0.000} C_DIS
LIN {X -9.724,Y -40.608,Z -77.623,A -90.000,B 90.000,C 0.000} C_DIS
LIN {X -9.252,Y -40.609,Z -77.625,A -90.000,B 90.000,C 0.000} C_DIS
LIN {X -9.100,Y -40.605,Z -77.627,A -90.000,B 90.000,C 0.000} C_DIS
LIN {X -8.482,Y -40.586,Z -77.637,A -90.000,B 90.000,C 0.000} C_DIS
LIN {X -8.397,Y -40.584,Z -77.640,A -90.000,B 90.000,C 0.000} C_DIS
LIN {X -6.115,Y -40.517,Z -77.805,A -90.000,B 90.000,C 0.000} C_DIS
LIN {X -5.327,Y -40.493,Z -77.868,A -90.000,B 90.000,C 0.000} C_DIS
LIN {X -5.226,Y -40.491,Z -77.879,A -90.000,B 90.000,C 0.000} C_DIS
LIN {X -4.700,Y -40.486,Z -77.946,A -90.000,B 90.000,C 0.000} C_DIS
LIN {X -3.200,Y -40.467,Z -78.170,A -90.000,B 90.000,C 0.000} C_DIS
LIN {X -1.780,Y -40.460,Z -78.424,A -90.000,B 90.000,C 0.000} C_DIS
LIN {X -1.130,Y -40.460,Z -78.547,A -90.000,B 90.000,C 0.000} C_DIS
LIN {X -0.246,Y -40.465,Z -78.723,A -90.000,B 90.000,C 0.000} C_DIS
LIN {X 1.347,Y -40.442,Z -79.057,A -90.000,B 90.000,C 0.000} C_DIS
LIN {X 2.016,Y -40.436,Z -79.205,A -90.000,B 90.000,C 0.000} C_DIS
LIN {X 4.326,Y -40.417,Z -79.713,A -90.000,B 90.000,C 0.000} C_DIS
LIN {X 5.631,Y -40.411,Z -80.022,A -90.000,B 90.000,C 0.000} C_DIS
LIN {X 6.992,Y -40.401,Z -80.348,A -90.000,B 90.000,C 0.000} C_DIS
LIN {X 8.528,Y -40.396,Z -80.733,A -90.000,B 90.000,C 0.000} C_DIS
LIN {X 10.211,Y -40.388,Z -81.157,A -90.000,B 90.000,C 0.000} C_DIS
LIN {X 11.103,Y -40.392,Z -81.403,A -90.000,B 90.000,C 0.000} C_DIS
LIN {X 11.691,Y -40.382,Z -81.548,A -90.000,B 90.000,C 0.000} C_DIS
LIN {X 12.013,Y -40.376,Z -81.626,A -90.000,B 90.000,C 0.000} C_DIS
LIN {X 13.040,Y -40.371,Z -81.874,A -90.000,B 90.000,C 0.000} C_DIS
LIN {X 13.967,Y -40.368,Z -82.126,A -90.000,B 90.000,C 0.000} C_DIS
LIN {X 14.722,Y -40.344,Z -82.289,A -90.000,B 90.000,C 0.000} C_DIS
LIN {X 14.830,Y -40.342,Z -82.311,A -90.000,B 90.000,C 0.000} C_DIS
LIN {X 16.634,Y -40.381,Z -82.682,A -90.000,B 90.000,C 0.000} C_DIS
LIN {X 16.946,Y -40.380,Z -82.727,A -90.000,B 90.000,C 0.000} C_DIS
LIN {X 17.451,Y -40.376,Z -82.794,A -90.000,B 90.000,C 0.000} C_DIS
LIN {X 18.030,Y -40.407,Z -82.851,A -90.000,B 90.000,C 0.000} C_DIS
LIN {X 19.008,Y -40.488,Z -82.935,A -90.000,B 90.000,C 0.000} C_DIS
LIN {X 19.321,Y -40.515,Z -82.958,A -90.000,B 90.000,C 0.000} C_DIS
LIN {X 19.892,Y -40.553,Z -82.958,A -90.000,B 90.000,C 0.000} C_DIS
LIN {X 20.611,Y -40.626,Z -82.950,A -90.000,B 90.000,C 0.000} C_DIS
LIN {X 20.952,Y -40.669,Z -82.921,A -90.000,B 90.000,C 0.000} C_DIS
LIN {X 21.429,Y -40.727,Z -82.863,A -90.000,B 90.000,C 0.000} C_DIS
LIN {X 22.171,Y -40.808,Z -82.719,A -90.000,B 90.000,C 0.000} C_DIS
LIN {X 22.486,Y -40.822,Z -82.554,A -90.000,B 90.000,C 0.000} C_DIS
LIN {X 22.830,Y -40.846,Z -82.373,A -90.000,B 90.000,C 0.000} C_DIS
LIN {X 22.962,Y -40.847,Z -82.258,A -90.000,B 90.000,C 0.000} C_DIS
LIN {X 23.850,Y -40.865,Z -81.524,A -90.000,B 90.000,C 0.000} C_DIS
LIN {X 23.963,Y -40.860,Z -81.417,A -90.000,B 90.000,C 0.000} C_DIS
LIN {X 24.949,Y -40.812,Z -80.485,A -90.000,B 90.000,C 0.000} C_DIS
LIN {X 25.012,Y -40.807,Z -80.428,A -90.000,B 90.000,C 0.000} C_DIS
LIN {X 25.116,Y -40.799,Z -80.343,A -90.000,B 90.000,C 0.000} C_DIS
LIN {X 25.358,Y -40.788,Z -80.166,A -90.000,B 90.000,C 0.000} C_DIS
LIN {X 25.540,Y -40.778,Z -80.040,A -90.000,B 90.000,C 0.000} C_DIS
LIN {X 26.111,Y -40.703,Z -79.660,A -90.000,B 90.000,C 0.000} C_DIS
LIN {X 26.299,Y -40.681,Z -79.541,A -90.000,B 90.000,C 0.000} C_DIS
LIN {X 26.346,Y -40.709,Z -79.498,A -90.000,B 90.000,C 0.000} C_DIS
LIN {X 26.166,Y -40.696,Z -79.476,A -90.000,B 90.000,C 0.000} C_DIS
LIN {X 25.213,Y -40.608,Z -79.351,A -90.000,B 90.000,C 0.000} C_DIS
LIN {X 24.898,Y -40.580,Z -79.308,A -90.000,B 90.000,C 0.000} C_DIS
LIN {X 24.632,Y -40.565,Z -79.255,A -90.000,B 90.000,C 0.000} C_DIS
LIN {X 24.426,Y -40.558,Z -79.202,A -90.000,B 90.000,C 0.000} C_DIS
LIN {X 24.261,Y -40.556,Z -79.142,A -90.000,B 90.000,C 0.000} C_DIS
LIN {X 24.109,Y -40.556,Z -79.079,A -90.000,B 90.000,C 0.000} C_DIS
LIN {X 24.053,Y -40.553,Z -79.055,A -90.000,B 90.000,C 0.000} C_DIS
LIN {X 23.842,Y -40.549,Z -78.949,A -90.000,B 90.000,C 0.000} C_DIS
LIN {X 22.507,Y -40.565,Z -78.195,A -90.000,B 90.000,C 0.000} C_DIS
LIN {X 22.309,Y -40.564,Z -78.081,A -90.000,B 90.000,C 0.000} C_DIS
LIN {X 22.211,Y -40.565,Z -78.022,A -90.000,B 90.000,C 0.000} C_DIS
LIN {X 22.089,Y -40.560,Z -77.937,A -90.000,B 90.000,C 0.000} C_DIS
LIN {X 21.931,Y -40.560,Z -77.815,A -90.000,B 90.000,C 0.000} C_DIS
LIN {X 21.808,Y -40.560,Z -77.712,A -90.000,B 90.000,C 0.000} C_DIS
LIN {X 21.677,Y -40.569,Z -77.586,A -90.000,B 90.000,C 0.000} C_DIS
LIN {X 21.554,Y -40.581,Z -77.457,A -90.000,B 90.000,C 0.000} C_DIS
LIN {X 21.445,Y -40.601,Z -77.325,A -90.000,B 90.000,C 0.000} C_DIS
LIN {X 21.402,Y -40.610,Z -77.271,A -90.000,B 90.000,C 0.000} C_DIS
LIN {X 21.304,Y -40.634,Z -77.140,A -90.000,B 90.000,C 0.000} C_DIS
LIN {X 21.053,Y -40.692,Z -76.796,A -90.000,B 90.000,C 0.000} C_DIS
LIN {X 20.985,Y -40.711,Z -76.695,A -90.000,B 90.000,C 0.000} C_DIS
LIN {X 20.857,Y -40.763,Z -76.466,A -90.000,B 90.000,C 0.000} C_DIS
LIN {X 20.815,Y -40.785,Z -76.372,A -90.000,B 90.000,C 0.000} C_DIS
LIN {X 20.730,Y -40.828,Z -76.160,A -90.000,B 90.000,C 0.000} C_DIS
LIN {X 20.693,Y -40.847,Z -76.043,A -90.000,B 90.000,C 0.000} C_DIS
LIN {X 20.669,Y -40.863,Z -75.954,A -90.000,B 90.000,C 0.000} C_DIS
LIN {X 20.642,Y -40.888,Z -75.821,A -90.000,B 90.000,C 0.000} C_DIS
LIN {X 20.628,Y -40.907,Z -75.711,A -90.000,B 90.000,C 0.000} C_DIS
LIN {X 20.612,Y -40.936,Z -75.550,A -90.000,B 90.000,C 0.000} C_DIS
LIN {X 20.603,Y -40.960,Z -75.399,A -90.000,B 90.000,C 0.000} C_DIS
LIN {X 20.603,Y -40.968,Z -75.329,A -90.000,B 90.000,C 0.000} C_DIS
LIN {X 20.611,Y -40.986,Z -75.176,A -90.000,B 90.000,C 0.000} C_DIS
LIN {X 20.625,Y -41.002,Z -75.059,A -90.000,B 90.000,C 0.000} C_DIS
LIN {X 20.644,Y -41.019,Z -74.954,A -90.000,B 90.000,C 0.000} C_DIS
LIN {X 20.676,Y -41.041,Z -74.795,A -90.000,B 90.000,C 0.000} C_DIS
LIN {X 20.709,Y -41.052,Z -74.664,A -90.000,B 90.000,C 0.000} C_DIS
